METHOD M_GetAbsPos : ST_3DPoint
VAR_INPUT
	pChildPos	: POINTER TO ST_3DPoint;
	eTargetRef 	: E_TargetRef;
	nParam1		: UINT;
 	nParam2		: UINT;
	nParam3		: USINT;
	nParam4		: USINT;
	nZLevel		: USINT;
END_VAR
VAR_OUTPUT
	nErrorId 	: ERRORID;
	lrAngle		: LREAL;
END_VAR
VAR
	stLocPos : ST_3DPoint;
END_VAR
IF eTargetRef = E_TargetRef.TARGETREF_TwoDimArray THEN
	stLocPos := P_stRelPosLB;
	
	IF nParam3 = 1 THEN	//Area1
		IF nArea1CountPoints = 0 THEN
			nErrorId := E_ErrorIdObjMgmt.ERRORID_InvalidDrypadArea;  //Error
			RETURN;
		END_IF
		//X-Position berechnen
		stLocPos.X := stLocPos.X + stArea1Point1.X + (stArea1Point2.X - stArea1Point1.X) / (nArea1IntermedPointsX + 1) * (nParam1 - 1);
		//Y-Position berechnen
		stLocPos.Y := stLocPos.Y + stArea1Point1.Y + (stArea1Point2.Y - stArea1Point1.Y) / (nArea1IntermedPointsY + 1) * (nParam2 - 1);		
	ELSIF nParam3 = 2 THEN	//Area2
		IF nArea2CountPoints = 0 THEN
			nErrorId := E_ErrorIdObjMgmt.ERRORID_InvalidDrypadArea;  //Error
			RETURN;
		END_IF
		//X-Position berechnen
		stLocPos.X := stLocPos.X + stArea2Point1.X + (stArea2Point2.X - stArea2Point1.X) / (nArea2IntermedPointsX + 1) * (nParam1 - 1);
		//Y-Position berechnen
		stLocPos.Y := stLocPos.Y + stArea2Point1.Y + (stArea2Point2.Y - stArea2Point1.Y) / (nArea2IntermedPointsY + 1) * (nParam2 - 1);		
	END_IF
	
	M_GetAbsPos := pParentTarget^.M_GetAbsPos(pChildPos := ADR(stLocPos), eTargetRef:= E_TargetRef.TARGETREF_LeftBottom,
													nParam1:= 0,
													nParam2:= 0, nParam3:= 0, nParam4:= 0, nZLevel:= 0,
													lrAngle => lrAngle, nErrorId=> nErrorId);
ELSE
	M_GetAbsPos := SUPER^.M_GetAbsPos(pChildPos := pChildPos, eTargetRef:= eTargetRef,
													nParam1:= nParam1,
													nParam2:= nParam2, nParam3:= nParam3, nParam4:= 0, nZLevel:= nZLevel,
													lrAngle => lrAngle, nErrorId=> nErrorId);	
END_IF
END_METHOD

METHOD M_GetAllProps : ERRORID
VAR_INPUT
	refCmdData : REFERENCE TO  ST_CmdData;
END_VAR
SUPER^.M_GetAllProps(refCmdData);
refCmdData.aHeader[2] := nNotifyId;

nCurrentPropIndex := nCurrentPropIndex + 1;
refCmdData.n32Data[nCurrentPropIndex] := REAL_TO_DINT(rZOffset);
nCurrentPropIndex := nCurrentPropIndex + 1;
refCmdData.n32Data[nCurrentPropIndex] := REAL_TO_DINT(stArea1Point1.X);
nCurrentPropIndex := nCurrentPropIndex + 1;
refCmdData.n32Data[nCurrentPropIndex] := REAL_TO_DINT(stArea1Point1.Y);
nCurrentPropIndex := nCurrentPropIndex + 1;
refCmdData.n32Data[nCurrentPropIndex] := REAL_TO_DINT(stArea1Point2.X);
nCurrentPropIndex := nCurrentPropIndex + 1;
refCmdData.n32Data[nCurrentPropIndex] := REAL_TO_DINT(stArea1Point2.Y);
nCurrentPropIndex := nCurrentPropIndex + 1;
refCmdData.n32Data[nCurrentPropIndex] := nArea1IntermedPointsX;
nCurrentPropIndex := nCurrentPropIndex + 1;
refCmdData.n32Data[nCurrentPropIndex] := nArea1IntermedPointsY;
nCurrentPropIndex := nCurrentPropIndex + 1;
refCmdData.n32Data[nCurrentPropIndex] := REAL_TO_DINT(stArea2Point1.X);
nCurrentPropIndex := nCurrentPropIndex + 1;
refCmdData.n32Data[nCurrentPropIndex] := REAL_TO_DINT(stArea2Point1.Y);
nCurrentPropIndex := nCurrentPropIndex + 1;
refCmdData.n32Data[nCurrentPropIndex] := REAL_TO_DINT(stArea2Point2.X);
nCurrentPropIndex := nCurrentPropIndex + 1;
refCmdData.n32Data[nCurrentPropIndex] := REAL_TO_DINT(stArea2Point2.Y);
nCurrentPropIndex := nCurrentPropIndex + 1;
refCmdData.n32Data[nCurrentPropIndex] := nArea2IntermedPointsX;
nCurrentPropIndex := nCurrentPropIndex + 1;
refCmdData.n32Data[nCurrentPropIndex] := nArea2IntermedPointsY;
nCurrentPropIndex := nCurrentPropIndex + 1;
refCmdData.n32Data[nCurrentPropIndex] := nGCodeTargetNr;
END_METHOD

METHOD M_ResetPosData
VAR_INPUT
END_VAR
nCurrentColArea1 := 0;
nCurrentRowArea1 := 0;
nCurrentColArea2 := 0;
nCurrentRowArea2 := 0;
END_METHOD

METHOD M_SetAllProps : ERRORID
VAR_INPUT
	refCmdData : REFERENCE TO  ST_CmdData;
END_VAR
//Basisproperties schreiben (0 bis 7)
M_SetAllProps := SUPER^.M_SetAllProps(refCmdData);

IF M_SetAllProps > 0 THEN	//Error beim setzen der Base-Parameter
	RETURN;
END_IF

nCurrentPropIndex := nCurrentPropIndex + 1;
nSpecPropIndex := nCurrentPropIndex; 
rZOffset := DINT_TO_REAL(refCmdData.n32Data[nCurrentPropIndex]);
nCurrentPropIndex := nCurrentPropIndex + 1;
stArea1Point1.X := DINT_TO_REAL(refCmdData.n32Data[nCurrentPropIndex]);
nCurrentPropIndex := nCurrentPropIndex + 1;
stArea1Point1.Y	:= DINT_TO_REAL(refCmdData.n32Data[nCurrentPropIndex]);
nCurrentPropIndex := nCurrentPropIndex + 1;
stArea1Point2.X := DINT_TO_REAL(refCmdData.n32Data[nCurrentPropIndex]);
nCurrentPropIndex := nCurrentPropIndex + 1;
stArea1Point2.Y := DINT_TO_REAL(refCmdData.n32Data[nCurrentPropIndex]);
nCurrentPropIndex := nCurrentPropIndex + 1;
nArea1IntermedPointsX := DINT_TO_UINT(refCmdData.n32Data[nCurrentPropIndex]);
nCurrentPropIndex := nCurrentPropIndex + 1;
nArea1IntermedPointsY := DINT_TO_UINT(refCmdData.n32Data[nCurrentPropIndex]);

nArea1CountPoints := (nArea1IntermedPointsX + 2) * (nArea1IntermedPointsY + 2);

nCurrentPropIndex := nCurrentPropIndex + 1; 
stArea2Point1.X	:= DINT_TO_REAL(refCmdData.n32Data[nCurrentPropIndex]);
nCurrentPropIndex := nCurrentPropIndex + 1;
stArea2Point1.Y	:= DINT_TO_REAL(refCmdData.n32Data[nCurrentPropIndex]);
nCurrentPropIndex := nCurrentPropIndex + 1;
stArea2Point2.X	:= DINT_TO_REAL(refCmdData.n32Data[nCurrentPropIndex]);
nCurrentPropIndex := nCurrentPropIndex + 1;
stArea2Point2.Y	:= DINT_TO_REAL(refCmdData.n32Data[nCurrentPropIndex]);
nCurrentPropIndex := nCurrentPropIndex + 1;
nArea2IntermedPointsX := DINT_TO_UINT(refCmdData.n32Data[nCurrentPropIndex]);
nCurrentPropIndex := nCurrentPropIndex + 1;
nArea2IntermedPointsY := DINT_TO_UINT(refCmdData.n32Data[nCurrentPropIndex]);

IF stArea2Point1.X <  stArea2Point2.X AND stArea2Point1.Y <  stArea2Point2.Y THEN
	nArea2CountPoints := (nArea2IntermedPointsX + 2) * (nArea2IntermedPointsY + 2);
ELSE
 	nArea2CountPoints := 0;
END_IF

nCurrentPropIndex := nCurrentPropIndex + 1;
nGCodeTargetNr := DINT_TO_UINT(refCmdData.n32Data[nCurrentPropIndex]);
nNoOfProps := nCurrentPropIndex + 1;
END_METHOD

METHOD M_SetSingleProp : ERRORID
VAR_INPUT
	refCmdData : REFERENCE TO  ST_CmdData;
END_VAR
IF nSpecPropIndex = refCmdData.aHeader[1] THEN
	rZOffset := DINT_TO_REAL(refCmdData.n32Data[0]);
ELSIF (nSpecPropIndex + 1) = refCmdData.aHeader[1] THEN
	stArea1Point1.X := DINT_TO_REAL(refCmdData.n32Data[0]);
ELSIF (nSpecPropIndex + 2) = refCmdData.aHeader[1] THEN
	stArea1Point1.Y := DINT_TO_REAL(refCmdData.n32Data[0]);
ELSIF (nSpecPropIndex + 3) = refCmdData.aHeader[1] THEN
	stArea1Point2.X := DINT_TO_REAL(refCmdData.n32Data[0]);
ELSIF (nSpecPropIndex + 4) = refCmdData.aHeader[1] THEN
	stArea1Point2.Y := DINT_TO_REAL(refCmdData.n32Data[0]);
ELSIF (nSpecPropIndex + 5) = refCmdData.aHeader[1] THEN
	nArea1IntermedPointsX := DINT_TO_UINT(refCmdData.n32Data[0]);
ELSIF (nSpecPropIndex + 6) = refCmdData.aHeader[1] THEN
	nArea1IntermedPointsY := DINT_TO_UINT(refCmdData.n32Data[0]);
ELSIF (nSpecPropIndex + 7) = refCmdData.aHeader[1] THEN
	stArea2Point1.X := DINT_TO_REAL(refCmdData.n32Data[0]);
ELSIF (nSpecPropIndex + 8) = refCmdData.aHeader[1] THEN
	stArea2Point1.Y := DINT_TO_REAL(refCmdData.n32Data[0]);
ELSIF (nSpecPropIndex + 9) = refCmdData.aHeader[1] THEN
	stArea2Point2.X := DINT_TO_REAL(refCmdData.n32Data[0]);
ELSIF (nSpecPropIndex + 10) = refCmdData.aHeader[1] THEN
	stArea2Point2.Y := DINT_TO_REAL(refCmdData.n32Data[0]);
ELSIF (nSpecPropIndex + 11) = refCmdData.aHeader[1] THEN
	nArea2IntermedPointsX := DINT_TO_UINT(refCmdData.n32Data[0]);
ELSIF (nSpecPropIndex + 12) = refCmdData.aHeader[1] THEN
	nArea2IntermedPointsY := DINT_TO_UINT(refCmdData.n32Data[0]);
ELSE
	M_SetSingleProp := SUPER^.M_SetSingleProp(refCmdData);
END_IF
END_METHOD

METHOD M_UpdateProcessData
VAR_INPUT
END_VAR
//Processdaten übetragen
aObjProcData[nNotifyId].nObjId := nObjectID;
aObjProcData[nNotifyId].n32Data[0] := nArea1CountPoints;
IF nCurrentColArea1 = 0 THEN
	aObjProcData[nNotifyId].n32Data[1] := 0;
ELSE
	aObjProcData[nNotifyId].n32Data[1] := (nArea1IntermedPointsX + 2) * (nCurrentRowArea1 - 1) + nCurrentColArea1;
END_IF

aObjProcData[nNotifyId].n32Data[2] := nArea2CountPoints;

IF nCurrentColArea2 = 0 THEN
	aObjProcData[nNotifyId].n32Data[3] := 0;
ELSE
	aObjProcData[nNotifyId].n32Data[3] := (nArea2IntermedPointsX + 2) * (nCurrentRowArea2 - 1) + nCurrentColArea2;
END_IF
END_METHOD

PROPERTY P_nGCodeTargetNr : UINT
GET
P_nGCodeTargetNr := nGCodeTargetNr;
END_GET
END_PROPERTY

PROPERTY P_nNotifyId : UINT
GET
P_nNotifyId := nNotifyId;
END_GET
SET
nNotifyId := P_nNotifyId;
END_SET
END_PROPERTY

END_FUNCTION_BLOCK

// ---- Objects/Targets/Active/FB_TipCleaner.TcPOU
FUNCTION_BLOCK FB_TipCleaner EXTENDS FB_ActiveTarget
VAR
	eBasicAction		: E_Action;
	eStripState			: E_OpClState;
	
	//Spec-Properties
	stFirstPoint		: ST_3DPoint;	//FirstPoint und LastPoint ergeben eine Linie
	stLastPoint			: ST_3DPoint;	//FirstPoint und LastPoint ergeben eine Linie
	nIntermedPoints		: USINT;		//Anzahl der Punkte auf der von FirstPoint und LastPoint gebildeten Linie
	
	nClosedPos			: UINT;			//Verschlussposition
	
	//****************************************Aktionvariablen****************************************************
	bActionLock			: ARRAY[50..150] OF BOOL;
	
	fbTipCleanerInit	: FB_TipCleanerInit;
	
	//Action: "OpenClose"
	bOpenClose			: BOOL;
	nStateA_OpenClose	: USINT;	//Statemachine von A_OpenClose();
	nOpenCloseMode		: USINT;	//0=Open, 1=Close

END_VAR

VAR PERSISTENT
	nCurrentPoint		: USINT;
END_VAR

IF bInitFB THEN
	bInitFB := FALSE;
	F_CreateLinkedListHnd( ADR( aNodes ), SIZEOF( aNodes ), hList );
	//Fehlerstruktur vorausfüllen
	stError.ObjectId := nObjectID;
	stError.HardwareGrp := E_HardwareGrp.Nothing;
	stError.POU := E_POU.POU_FB_TipCleaner;
END_IF

CASE eCurrentState OF
	E_MachineState.MACHINESTATE_Active:
		//BasicActions ausführen
		IF bInit THEN	//Initialisieren
			A_Init();
			IF nStateA_Init >= 80 THEN
				bIsInit := TRUE;
				IF nStateA_Init >= 99 THEN
					bError := TRUE;
					bIsInit := FALSE;	
				END_IF
				bInit := FALSE;
				nStateA_Init := 0;
				M_RemoveListEntry(nSearchValue:= E_Action.ACTION_Init);
			END_IF
		END_IF
		
		IF bOpenClose THEN	//Backen auf/zu
			A_OpenClose();
			IF nStateA_OpenClose >= 80 THEN
				IF nStateA_OpenClose >= 99 THEN
					bError := TRUE;	
				END_IF
				bOpenClose := FALSE;
				nStateA_OpenClose := 0;
				M_RemoveListEntry(nSearchValue:= E_Action.ACTION_OpenClose);
			END_IF
		END_IF		

		IF hList.nCount = 0 THEN
			eCurrentState := E_MachineState.MACHINESTATE_Ready;
		END_IF

		IF bError  THEN
			eCurrentState := E_MachineState.MACHINESTATE_Error;
		END_IF		
	
	E_MachineState.MACHINESTATE_Reset:
		A_Reset();
		IF nStateA_Reset = 80 THEN
			nStateA_Init := 0;
			nStateA_OpenClose := 0;
			nStateA_Stop := 0;
			nStateA_Reset := 0;
			bBusy := FALSE;
			bError := FALSE;
			bStopAllOnError := FALSE;
			fbList.A_Reset(hList := hList);
			MEMSET(ADR(bActionLock),0,SIZEOF(bActionLock));
			nErrorId := 0;
			stError.Cmd := 0;
			stError.ErrorId := 0;
			eCurrentState := E_MachineState.MACHINESTATE_Idle;
		ELSIF
			nStateA_Reset = 99 THEN
			fbErrorList.M_Add(stError);
			nStateA_Reset := 0;
			bBusy := FALSE;
			bError := TRUE;
			eCurrentState := E_MachineState.MACHINESTATE_Error;			
		END_IF
	
	E_MachineState.MACHINESTATE_Ready:
		bBusy := FALSE;
		eCurrentState := E_MachineState.MACHINESTATE_Idle;
		
	E_MachineState.MACHINESTATE_Error:
		bBusy := FALSE;	
	
END_CASE

//Prozessdaten aktualisieren
stProcessData.nObjId := nObjectID;
stProcessData.n32Data[0] := BOOL_TO_DINT(bIsInit);
stProcessData.n32Data[1] := eCurrentState;
stProcessData.n32Data[2] := stError.ErrorId;
IF stTipCleanerRef.nCurrentPos = 0 THEN
	eStripState := E_OpClState.Open;
	stProcessData.n32Data[3] := E_OpClState.Open;
ELSIF stTipCleanerRef.nCurrentPos = nClosedPos THEN
		eStripState := E_OpClState.Closed;
	stProcessData.n32Data[3] := E_OpClState.Closed;
ELSE
	eStripState := E_OpClState.UNDEFINED;
	stProcessData.n32Data[3] := E_OpClState.UNDEFINED;
END_IF

stProcessData.n32Data[4] := nIntermedPoints + 2; //Konfigurierte Reinigungspositionen
stProcessData.n32Data[5] := nCurrentPoint;	//verbrauchte Reinigungspositionen

aObjProcData[nNotifyId] := stProcessData;

ACTION A_Init:
IF nStateA_Init = 0 THEN
	bIsInit := FALSE;

	IF bFlagA_Init XOR fbTipCleanerInit.bBusy  THEN
		bFlagA_Init := FALSE;
		fbTipCleanerInit(pstTipCleanerRef:= ADR(stTipCleanerRef), bExecute:= TRUE);
	ELSE
		RETURN;	//damit nachfolgende Zeilen nicht bearbeitet werden
	END_IF		

	IF NOT fbTipCleanerInit.bBusy THEN
		IF fbTipCleanerInit.bError THEN
			stError.ErrorId := fbTipCleanerInit.nErrorId;
			stError.POUState := nStateA_Init;
			nStateA_Init := 99;
		ELSE
			bFlagA_Init := TRUE;
			nStateA_Init := 80;
		END_IF
		fbTipCleanerInit(pstTipCleanerRef:= ADR(stTipCleanerRef), bExecute:= FALSE);
	END_IF
END_IF

//Errorhandling
IF nStateA_Init = 99 THEN
	stError.Cmd := E_Action.ACTION_Init;
	stError.POUAction := E_POUACT.POUACT_A_Init;
	fbErrorList.M_Add(stError);
END_IF
END_ACTION

ACTION A_OpenClose:
stError.POUState := nStateA_OpenClose;

IF stTipCleanerRef.nStatus.3 THEN	//Error
	stError.ErrorId := E_ErrorIdCmd.ERRORID_DeviceInErrorState;
	nStateA_OpenClose := 99;
END_IF

CASE nStateA_OpenClose OF
	0:
		IF nOpenCloseMode = 0 THEN	//Öffnen
			stTipCleanerRef.nTargetPos := 0;
		ELSE	//Schließen
			stTipCleanerRef.nTargetPos := nClosedPos;
		END_IF
		
		stTipCleanerRef.nControl := 31;
		
		IF stTipCleanerRef.nStatus.12 THEN	//Setpoint acknowledge
			stTipCleanerRef.nControl := 15;
			nStateA_OpenClose := 1;
		END_IF
		
	1:	//Warten auf Target reached
		IF stTipCleanerRef.nStatus.10 THEN	//Target reached
			nStateA_OpenClose := 80;
		END_IF
		
	70:	//Cancel
		nStateA_OpenClose := 80;
END_CASE

//Errorhandling
IF nStateA_OpenClose = 99 THEN
	stError.Cmd := E_Action.ACTION_OpenClose;
	stError.POUAction := E_POUACT.POUACT_A_OpenClose;
	fbErrorList.M_Add(stError);
END_IF
END_ACTION

ACTION A_Reset:
CASE nStateA_Reset OF
	0:
		nStateA_Reset := 80;
END_CASE
END_ACTION

METHOD FB_init : BOOL
VAR_INPUT
	bInitRetains : BOOL; // if TRUE, the retain variables are initialized (warm start / cold start)
	bInCopyCode : BOOL;  // if TRUE, the instance afterwards gets moved into the copy code (online change)
END_VAR
eObjectType := E_ObjectType.OBJECTTYPE_TipCleaner;
eObjectGroup := E_ObjectGroup.OBJECTGROUP_Target OR E_ObjectGroup.OBJECTGROUP_Device;
END_METHOD

METHOD M_ChangeCleanMat
VAR_INPUT
END_VAR
nCurrentPoint := 0;
END_METHOD

METHOD M_CheckAction : ERRORID
VAR_INPUT
	refActionData 	: REFERENCE TO ST_ActionData;
	pCorrelObject	: POINTER TO FB_Object;
END_VAR
IF NOT refActionData.eAction = E_Action.ACTION_MoveToTarget THEN
	M_CheckAction := 8989;	
END_IF
END_METHOD

METHOD M_CheckProcDataType : BOOL
VAR_INPUT
	eProcDataType : E_ProcDataType;
END_VAR
END_METHOD

METHOD M_ExeAction : ERRORID
VAR_INPUT
	refActionData : REFERENCE TO ST_ActionData;	
END_VAR
IF NOT (eCurrentState = E_MachineState.MACHINESTATE_Idle OR
	eCurrentState = E_MachineState.MACHINESTATE_Active OR
	eCurrentState = E_MachineState.MACHINESTATE_Ready) THEN
	M_ExeAction := E_ErrorIdCmd.ERRORID_InvalidState;
	RETURN;
END_IF

CASE refActionData.eAction OF
	E_Action.ACTION_Init:
		IF NOT bInit THEN
			bInit := TRUE;
			fbList.A_AddHeadValue(hList := hList, putValue:= E_Action.ACTION_Init);
		ELSE
			RETURN;
		END_IF
		
	E_Action.ACTION_OpenClose:
		IF NOT bOpenClose THEN
			IF NOT bIsInit THEN
				M_ExeAction := E_ErrorIdCmd.ERRORID_DeviceNotInitialized;  //Error
				RETURN;
			END_IF
			nOpenCloseMode := DINT_TO_USINT(refActionData.aParams[1]);
			fbList.A_AddHeadValue(hList := hList, putValue:= E_Action.ACTION_OpenClose);
			bOpenClose := TRUE;
		ELSE
			RETURN;
		END_IF
		
	E_Action.ACTION_Stop:
		//Stop braucht nur ausgeführt werden, wenn irgendwas aktiv ist
		fbList.A_AddHeadValue(hList := hList, putValue:= E_Action.ACTION_Stop);		
	ELSE
		M_ExeAction := E_ErrorIdCmd.ERRORID_InvalidAction;
END_CASE
bBusy := TRUE;
eCurrentState := E_MachineState.MACHINESTATE_Active;
END_METHOD

METHOD M_GetAbsPos : ST_3DPoint
VAR_INPUT
	pChildPos	: POINTER TO ST_3DPoint;
	eTargetRef 	: E_TargetRef;
	nParam1		: UINT;
 	nParam2		: UINT;
	nParam3		: USINT;
	nParam4		: USINT;
	nZLevel		: USINT;
END_VAR
VAR_OUTPUT
	nErrorId 	: ERRORID;
	lrAngle		: LREAL;
END_VAR
VAR
	stLocPosLB : ST_3DPoint;
	rSpace	: REAL;
END_VAR
IF eTargetRef = E_TargetRef.TARGETREF_SpecPoint THEN
	stLocPosLB := P_stRelPosLB;
	IF nParam1 = 1 THEN
		stLocPosLB := F_Add3DPoints(stLocPosLB,stFirstPoint);
	ELSIF nParam1 = 2 THEN
		stLocPosLB := F_Add3DPoints(stLocPosLB,stLastPoint);
	ELSE
		nErrorId := E_ErrorIdCmd.ERRORID_InvalidTargetPointNr;
		RETURN;
	END_IF
	M_GetAbsPos := pParentTarget^.M_GetAbsPos(pChildPos := ADR(stLocPosLB), eTargetRef:= E_TargetRef.TARGETREF_LeftBottom,
												nParam1:= 0,
												nParam2:= 0, nParam3:= 0, nParam4:= 0, nZLevel:= 0,
												lrAngle => lrAngle, nErrorId=> nErrorId);	
ELSIF eTargetRef = E_TargetRef.TARGETREF_TwoDimArray THEN
	//Checken ob gültiger Punkt
	IF nParam1 = 0 OR nParam1 > (nIntermedPoints + 2) THEN
		nErrorId := E_ErrorIdCmd.ERRORID_InvalidTargetPointCol;
		RETURN;
	END_IF
	stLocPosLB := P_stRelPosLB;
	//Ausrichtung in X oder Y?
	IF stFirstPoint.Y = stLastPoint.Y THEN	//Ausrichtung in X
		//X-Position berechnen
		//Space(Zwischenräume zwischen den Punkten berechnen
		rSpace := (stLastPoint.X - stFirstPoint.X) / (nIntermedPoints + 1); 
		stLocPosLB.X := stLocPosLB.X + stFirstPoint.X + (nParam1 - 1) * rSpace;
		//Y-Position berechenen
		stLocPosLB.Y := stLocPosLB.Y + stFirstPoint.Y;
	ELSIF stFirstPoint.X = stLastPoint.X THEN //Ausrichtung in Y
		//X-Position berechnen
		stLocPosLB.X := stLocPosLB.X + stFirstPoint.X;
		//Y-Position berechenen
		//Space(Zwischenräume zwischen den Punkten berechnen
		rSpace := (stLastPoint.Y - stFirstPoint.Y) / (nIntermedPoints + 1);
		stLocPosLB.Y := stLocPosLB.Y + stFirstPoint.Y + (nParam1 - 1) * rSpace;
	ELSE
		nErrorId := E_ErrorIdCmd.ERRORID_InvalidTargetPointCol;
		RETURN;
	END_IF
	stLocPosLB.Z := stLocPosLB.Z + stFirstPoint.Z;
	M_GetAbsPos := pParentTarget^.M_GetAbsPos(pChildPos := ADR(stLocPosLB), eTargetRef:= E_TargetRef.TARGETREF_LeftBottom,
												nParam1:= 0,
												nParam2:= 0, nParam3:= 0,nParam4:= 0, nZLevel:= 0,
												lrAngle => lrAngle, nErrorId=> nErrorId);	

ELSE
	M_GetAbsPos := SUPER^.M_GetAbsPos(pChildPos := pChildPos, eTargetRef:= eTargetRef,
													nParam1:= nParam1,
													nParam2:= nParam2, nParam3:= nParam3, nParam4:= 0, nZLevel:= nZLevel,
													lrAngle => lrAngle, nErrorId=> nErrorId);	
END_IF
END_METHOD

METHOD M_GetActionBusy : BOOL
VAR_INPUT
	eAction : E_Action;
END_VAR
getPosPtr := 0;(* start from first node element *)
fbList.A_FindNext( hList := hList, putPosPtr := getPosPtr, putValue := eAction, getValue=>getValue, getPosPtr=>getPosPtr );
IF fbList.bOk THEN	//Eintrag wurde gefunden, d.h. Action ist noch busy
	M_GetActionBusy := TRUE;
END_IF
END_METHOD

METHOD M_GetAllProps : ERRORID
VAR_INPUT
	refCmdData : REFERENCE TO  ST_CmdData;
END_VAR
SUPER^.M_GetAllProps(refCmdData);
nCurrentPropIndex := nCurrentPropIndex + 1;
refCmdData.n32Data[nCurrentPropIndex] := REAL_TO_DINT(stFirstPoint.X);
nCurrentPropIndex := nCurrentPropIndex + 1;
refCmdData.n32Data[nCurrentPropIndex] := REAL_TO_DINT(stFirstPoint.Y);
nCurrentPropIndex := nCurrentPropIndex + 1;
refCmdData.n32Data[nCurrentPropIndex] := REAL_TO_DINT(stFirstPoint.Z);
nCurrentPropIndex := nCurrentPropIndex + 1;
refCmdData.n32Data[nCurrentPropIndex] := REAL_TO_DINT(stLastPoint.X);
nCurrentPropIndex := nCurrentPropIndex + 1;
refCmdData.n32Data[nCurrentPropIndex] := REAL_TO_DINT(stLastPoint.Y);
nCurrentPropIndex := nCurrentPropIndex + 1;
refCmdData.n32Data[nCurrentPropIndex] := nIntermedPoints;
nCurrentPropIndex := nCurrentPropIndex + 1;
refCmdData.n32Data[nCurrentPropIndex] := nClosedPos;
END_METHOD

METHOD M_GetNextPointNr : USINT
VAR_INPUT
END_VAR
IF (nCurrentPoint = (nIntermedPoints + 2)) OR (nCurrentPoint = 0) THEN
	nCurrentPoint := 1;
ELSE
	nCurrentPoint := nCurrentPoint + 1;
END_IF
M_GetNextPointNr := nCurrentPoint;
END_METHOD

METHOD M_GetProcData : DINT
VAR_INPUT
	eProcDataType : E_ProcDataType;
END_VAR
END_METHOD

METHOD M_RemoveListEntry : BOOL
VAR_INPUT
	nSearchValue	: E_Action;
END_VAR
getPosPtr := 0;(* start from first node element *)
fbList.A_FindNext( hList := hList, putPosPtr := getPosPtr, putValue := nSearchValue, getValue=>getValue, getPosPtr=>getPosPtr );
IF fbList.bOk THEN	//Eintrag wurde gefunden
	fbList.A_RemoveValueAtPosPtr(hList:= hList,	putPosPtr:= getPosPtr);
	IF fbList.bOk THEN
		M_RemoveListEntry := TRUE;
	END_IF
END_IF
END_METHOD

METHOD M_SetAllProps : ERRORID
VAR_INPUT
	refCmdData : REFERENCE TO  ST_CmdData;
END_VAR
M_SetAllProps := SUPER^.M_SetAllProps(refCmdData);

IF M_SetAllProps > 0 THEN
	RETURN;
END_IF

nCurrentPropIndex := nCurrentPropIndex + 1;
nSpecPropIndex := nCurrentPropIndex;
stFirstPoint.X := DINT_TO_REAL(refCmdData.n32Data[nCurrentPropIndex]);
nCurrentPropIndex := nCurrentPropIndex + 1;
stFirstPoint.Y := DINT_TO_REAL(refCmdData.n32Data[nCurrentPropIndex]);
nCurrentPropIndex := nCurrentPropIndex + 1;
stFirstPoint.Z := DINT_TO_REAL(refCmdData.n32Data[nCurrentPropIndex]);
nCurrentPropIndex := nCurrentPropIndex + 1; 
stLastPoint.X := DINT_TO_REAL(refCmdData.n32Data[nCurrentPropIndex]);
nCurrentPropIndex := nCurrentPropIndex + 1;
stLastPoint.Y := DINT_TO_REAL(refCmdData.n32Data[nCurrentPropIndex]);
stLastPoint.Z := stFirstPoint.Z;
nCurrentPropIndex := nCurrentPropIndex + 1;
nIntermedPoints := DINT_TO_USINT(refCmdData.n32Data[nCurrentPropIndex]);
nCurrentPropIndex := nCurrentPropIndex + 1;
nClosedPos := DINT_TO_UINT(refCmdData.n32Data[nCurrentPropIndex]);

nNoOfProps := nCurrentPropIndex + 1;
END_METHOD

METHOD M_SetSingleProp : ERRORID
VAR_INPUT
	refCmdData : REFERENCE TO  ST_CmdData;
END_VAR
IF nSpecPropIndex = refCmdData.aHeader[1] THEN
	stFirstPoint.X := DINT_TO_REAL(refCmdData.n32Data[0]);
ELSIF (nSpecPropIndex + 1) = refCmdData.aHeader[1] THEN
	stFirstPoint.Y := DINT_TO_REAL(refCmdData.n32Data[0]);
ELSIF (nSpecPropIndex + 2) = refCmdData.aHeader[1] THEN
	stFirstPoint.Z := DINT_TO_REAL(refCmdData.n32Data[0]);
ELSIF (nSpecPropIndex + 3) = refCmdData.aHeader[1] THEN
	stLastPoint.X := DINT_TO_REAL(refCmdData.n32Data[0]);
ELSIF (nSpecPropIndex + 4) = refCmdData.aHeader[1] THEN
	stLastPoint.Y := DINT_TO_REAL(refCmdData.n32Data[0]);
ELSIF (nSpecPropIndex + 5) = refCmdData.aHeader[1] THEN
	nIntermedPoints := DINT_TO_USINT(refCmdData.n32Data[0]);
ELSIF (nSpecPropIndex + 6) = refCmdData.aHeader[1] THEN
	nClosedPos := DINT_TO_UINT(refCmdData.n32Data[0]);	
ELSE
	M_SetSingleProp := SUPER^.M_SetSingleProp(refCmdData);
END_IF
END_METHOD

METHOD M_Stop : ERRORID
VAR_INPUT
END_VAR
IF bOpenClose THEN
	nStateA_OpenClose := 70;
END_IF
END_METHOD

PROPERTY P_eStripState : E_OpClState
GET
P_eStripState := eStripState;
END_GET
END_PROPERTY

END_FUNCTION_BLOCK

// ---- Hardware/TipCleaner/FB_TipCleanerInit.TcPOU
FUNCTION_BLOCK FB_TipCleanerInit
VAR_INPUT
	pstTipCleanerRef	: POINTER TO ST_TipCleanerRef;
	bExecute			: BOOL;
END_VAR
VAR_OUTPUT
	bBusy		: BOOL;
	bError		: BOOL;
	nErrorId	: ERRORID;
END_VAR
VAR
	fbSdoWrite	: FB_SDO_WRITE;
	nIndex		: DWORD;
	nSubIndex	: DWORD;
	nDataLength	: DWORD;
	nData		: DINT;
	nState		: USINT;
	timer		: TON;
END_VAR

IF bExecute THEN
	bBusy := TRUE;
	CASE nState OF
		0:	//*************ANFANG INITIALISIERUNG ************************************
			IF pstTipCleanerRef^.nStatus.3 THEN	//Error?
				pstTipCleanerRef^.nControl := 153;	//Error zurücksetzen
			ELSE
				pstTipCleanerRef^.nControl := 0;
				nState := nState + 1;
			END_IF
			
		1:	//max Strom auf 0,8A begrenzen (TMCM1140 max 2A entspricht "255" in Object 0x2003)
			fbSdoWrite(sADSNetID:= pstTipCleanerRef^.stAdsAdress.sNetId,nPortNr:= pstTipCleanerRef^.stAdsAdress.nPort, 
						nIndex:= 16#2003, nSubIndex:= 0, nDataLength:= 1, nData:= 128, bExecute:= TRUE);
			 	
			IF NOT fbSdoWrite.bBusy THEN
				IF fbSdoWrite.bError THEN
					nErrorId := fbSdoWrite.nAdsErrorId;
					nState := 99;
				ELSE
					nState := nState + 1;
				END_IF
				fbSdoWrite(bExecute:= FALSE);
			END_IF

		2:	//Standby Strom auf 0,2A begrenzen (TMCM1140 max 2A entspricht "255" in Object 0x2004)
			(*fbSdoWrite(sADSNetID:= pstTipCleanerRef^.stAdsAdress.sNetId,nPortNr:= pstTipCleanerRef^.stAdsAdress.nPort, 
						nIndex:= 16#2004, nSubIndex:= 0, nDataLength:= 1, nData:= 35, bExecute:= TRUE);*)
			 	
			fbSdoWrite(sADSNetID:= pstTipCleanerRef^.stAdsAdress.sNetId,nPortNr:= pstTipCleanerRef^.stAdsAdress.nPort, 
						nIndex:= 16#2004, nSubIndex:= 0, nDataLength:= 1, nData:= 0, bExecute:= TRUE);

			IF NOT fbSdoWrite.bBusy THEN
				IF fbSdoWrite.bError THEN
					nErrorId := fbSdoWrite.nAdsErrorId;
					nState := 99;
				ELSE
					nState := nState + 1;
				END_IF
				fbSdoWrite(bExecute:= FALSE);
			END_IF
			
		3:	//SwitchParameters setzen (keine Endlagen verwenden)
			fbSdoWrite(sADSNetID:= pstTipCleanerRef^.stAdsAdress.sNetId,nPortNr:= pstTipCleanerRef^.stAdsAdress.nPort, 
						nIndex:= 16#2005, nSubIndex:= 0, nDataLength:= 4, nData:= 3, bExecute:= TRUE);
			 	
			IF NOT fbSdoWrite.bBusy THEN
				IF fbSdoWrite.bError THEN
					nErrorId := fbSdoWrite.nAdsErrorId;
					nState := 99;
				ELSE
					nState := nState + 1;
				END_IF
				fbSdoWrite(bExecute:= FALSE);
			END_IF

		4:	//Brake deaktivieren
			fbSdoWrite(sADSNetID:= pstTipCleanerRef^.stAdsAdress.sNetId,nPortNr:= pstTipCleanerRef^.stAdsAdress.nPort, 
						nIndex:= 16#200C, nSubIndex:= 2, nDataLength:= 1, nData:= 0, bExecute:= TRUE);

			IF NOT fbSdoWrite.bBusy THEN
				IF fbSdoWrite.bError THEN
					nErrorId := fbSdoWrite.nAdsErrorId;
					nState := 99;
				ELSE
					nState := nState + 1;
				END_IF
				fbSdoWrite(bExecute:= FALSE);
			END_IF
			
		5:	//Digital Outputmask setzen
			fbSdoWrite(sADSNetID:= pstTipCleanerRef^.stAdsAdress.sNetId,nPortNr:= pstTipCleanerRef^.stAdsAdress.nPort, 
						nIndex:= 16#2703, nSubIndex:= 2, nDataLength:= 4, nData:= 16#30000, bExecute:= TRUE);

			IF NOT fbSdoWrite.bBusy THEN
				IF fbSdoWrite.bError THEN
					nErrorId := fbSdoWrite.nAdsErrorId;
					nState := 99;
				ELSE
					nState := nState + 1;
				END_IF
				fbSdoWrite(bExecute:= FALSE);
			END_IF

		6:	//Fast Homing Speed setzen
			fbSdoWrite(sADSNetID:= pstTipCleanerRef^.stAdsAdress.sNetId,nPortNr:= pstTipCleanerRef^.stAdsAdress.nPort, 
						nIndex:= 16#6099, nSubIndex:= 1, nDataLength:= 4, nData:= 200, bExecute:= TRUE);

			IF NOT fbSdoWrite.bBusy THEN
				IF fbSdoWrite.bError THEN
					nErrorId := fbSdoWrite.nAdsErrorId;
					nState := 99;
				ELSE
					nState := nState + 1;
				END_IF
				fbSdoWrite(bExecute:= FALSE);
			END_IF

		7:	//Slow Homing Speed setzen
			fbSdoWrite(sADSNetID:= pstTipCleanerRef^.stAdsAdress.sNetId,nPortNr:= pstTipCleanerRef^.stAdsAdress.nPort, 
						nIndex:= 16#6099, nSubIndex:= 2, nDataLength:= 4, nData:= 100, bExecute:= TRUE);

			IF NOT fbSdoWrite.bBusy THEN
				IF fbSdoWrite.bError THEN
					nErrorId := fbSdoWrite.nAdsErrorId;
					nState := 99;
				ELSE
					nState := nState + 1;
				END_IF
				fbSdoWrite(bExecute:= FALSE);
			END_IF
			
		8:	//Profile Velo setzen
			fbSdoWrite(sADSNetID:= pstTipCleanerRef^.stAdsAdress.sNetId,nPortNr:= pstTipCleanerRef^.stAdsAdress.nPort, 
						nIndex:= 16#6081, nSubIndex:= 0, nDataLength:= 4, nData:= 800, bExecute:= TRUE);

			IF NOT fbSdoWrite.bBusy THEN
				IF fbSdoWrite.bError THEN
					nErrorId := fbSdoWrite.nAdsErrorId;
					nState := 99;
				ELSE
					nState := nState + 1;
				END_IF
				fbSdoWrite(bExecute:= FALSE);
			END_IF

		9:	//Homing Method setzen
			fbSdoWrite(sADSNetID:= pstTipCleanerRef^.stAdsAdress.sNetId,nPortNr:= pstTipCleanerRef^.stAdsAdress.nPort, 
						nIndex:= 16#6098, nSubIndex:= 0, nDataLength:= 1, nData:= 19, bExecute:= TRUE);

			IF NOT fbSdoWrite.bBusy THEN
				IF fbSdoWrite.bError THEN
					nErrorId := fbSdoWrite.nAdsErrorId;
					nState := 99;
				ELSE
					nState := nState + 1;
				END_IF
				fbSdoWrite(bExecute:= FALSE);
			END_IF
			
		10:	//Position Window setzen
			fbSdoWrite(sADSNetID:= pstTipCleanerRef^.stAdsAdress.sNetId,nPortNr:= pstTipCleanerRef^.stAdsAdress.nPort, 
						nIndex:= 16#6067, nSubIndex:= 0, nDataLength:= 4, nData:= 100, bExecute:= TRUE);

			IF NOT fbSdoWrite.bBusy THEN
				IF fbSdoWrite.bError THEN
					nErrorId := fbSdoWrite.nAdsErrorId;
					nState := 99;
				ELSE
					nState := nState + 1;
				END_IF
				fbSdoWrite(bExecute:= FALSE);
			END_IF
			
		11:	//Leistungsteil einschalten - "Ready to switch on"
			pstTipCleanerRef^.nControl := 6;
			pstTipCleanerRef^.bVDD5V := TRUE;	//Versorgung für Digitale IOs (5V) einschalten
			nState := nState + 1;

		12:	//Abfrage auf Status "Ready to switch on"
			IF F_GetCoDS402State(pstTipCleanerRef^.nStatus) = E_CoDS402States.DS402STATE_Fault THEN  //Error
				nState := 99;
			ELSIF F_GetCoDS402State(pstTipCleanerRef^.nStatus) = E_CoDS402States.DS402STATE_ReadyToSwitchOn  THEN//"Ready to switch on"
				nState := nState + 1;
			END_IF

		13:	//Leistungsteil einschalten - "Switch on" und "Voltage Enabled"
			pstTipCleanerRef^.nControl := 7;
			nState := nState + 1;
			
		14:	//Abfrage auf Status "Switch on" und "Voltage Enabled"
			IF F_GetCoDS402State(pstTipCleanerRef^.nStatus) = E_CoDS402States.DS402STATE_Fault THEN  //Error
				nState := 99;
			ELSIF F_GetCoDS402State(pstTipCleanerRef^.nStatus) = E_CoDS402States.DS402STATE_SwitchedOn THEN //"Switch on" und "Voltage Enabled"
				nState := nState + 1;
			END_IF

		15:	//Leistungsteil einschalten - "Operation Enabled"
			pstTipCleanerRef^.nControl := 15;
			nState := nState + 1;

		16:	//Abfrage auf Status "Operation Enabled"
			IF F_GetCoDS402State(pstTipCleanerRef^.nStatus) = E_CoDS402States.DS402STATE_Fault THEN  //Error
				nState := 99;
			ELSIF F_GetCoDS402State(pstTipCleanerRef^.nStatus) = E_CoDS402States.DS402STATE_OperationEnabled THEN //"Operation Enabled"
				nState := nState + 1;
			END_IF
			
		17:	//Mode of Operation auf "Homing" setzen
			pstTipCleanerRef^.nMode := 6;
			IF pstTipCleanerRef^.nModeDisp = 6 THEN
				nState := nState + 1;
			END_IF
			
		18:	//Homing Starten
			pstTipCleanerRef^.nControl := 31;
			IF pstTipCleanerRef^.nStatus.3 OR pstTipCleanerRef^.nStatus.13 THEN //Error
				nState := 99;
			ELSIF NOT pstTipCleanerRef^.nStatus.10 AND NOT pstTipCleanerRef^.nStatus.12 AND NOT pstTipCleanerRef^.nStatus.13 THEN	//Homig in process
				nState := nState + 1;
				timer(IN:= FALSE);
			END_IF
			
		19:	//Homing ready?
			timer(IN:= TRUE, PT:=T#6S);
			IF timer.Q THEN	//Error
				timer(IN:= FALSE);
				pstTipCleanerRef^.nControl := 0;
				nState := 99;
				RETURN;
			END_IF
			
			IF pstTipCleanerRef^.nStatus.3 OR pstTipCleanerRef^.nStatus.13 THEN //Error
				nState := 99;
			ELSIF pstTipCleanerRef^.nStatus.10 AND pstTipCleanerRef^.nStatus.12 AND NOT pstTipCleanerRef^.nStatus.13 THEN
				pstTipCleanerRef^.nControl := 15;
				nState := nState + 1;
			END_IF

		20:	//Mode of Operation auf "PP" setzen
			pstTipCleanerRef^.nMode := 1;
			IF pstTipCleanerRef^.nModeDisp = 1 THEN
				nState := nState + 1;
				bBusy := FALSE;
			END_IF

		99:	//Error
			bBusy := FALSE;
			bError := TRUE;
	END_CASE
 ELSE
	bError := FALSE;
	nErrorId := 0;
	nState := 0;
END_IF

END_FUNCTION_BLOCK

// ---- Hardware/F_GetCoDS402State.TcPOU
FUNCTION F_GetCoDS402State : E_CoDS402States
VAR_INPUT
	nStatus	: UINT;
END_VAR
VAR
	nStatusTemp	: UINT;
END_VAR

IF (nStatus AND 16#4F) = 0 THEN
	F_GetCoDS402State := E_CoDS402States.DS402STATE_NotReadyToSwitchOn;
ELSIF (nStatus AND 16#4F) = 16#40 THEN
	F_GetCoDS402State := E_CoDS402States.DS402STATE_SwitchOnDisabled;
ELSIF (nStatus AND 16#6F) = 16#21 THEN
	F_GetCoDS402State := E_CoDS402States.DS402STATE_ReadyToSwitchOn;
ELSIF (nStatus AND 16#6F) = 16#23 THEN
	F_GetCoDS402State := E_CoDS402States.DS402STATE_SwitchedOn;
ELSIF (nStatus AND 16#6F) = 16#27 THEN
	F_GetCoDS402State := E_CoDS402States.DS402STATE_OperationEnabled;
ELSIF (nStatus AND 16#6F) = 16#07 THEN
	F_GetCoDS402State := E_CoDS402States.DS402STATE_QuickStopActive;
ELSIF (nStatus AND 16#1400) = 16#1400 THEN
	F_GetCoDS402State := E_CoDS402States.DS402STATE_HomingCompleted;
ELSIF (nStatus AND 16#4F) = 16#0F THEN
	F_GetCoDS402State := E_CoDS402States.DS402STATE_FaultReactionActive;
ELSIF (nStatus AND 16#4F) = 16#08 THEN
	F_GetCoDS402State := E_CoDS402States.DS402STATE_Fault;
ELSE
	F_GetCoDS402State := E_CoDS402States.DS402STATE_Notspecified;
END_IF

END_FUNCTION

// ---- MainProgs/PC_Control.TcPOU
PROGRAM PC_Control
VAR
	fbWriteInd  	: ADSWRITEIND;
	fbWriteRes  	: ADSWRITERES;
	fbReadInd		: ADSREADIND;
	fbReadRes		: ADSREADRES;
	fbReadWriteInd	: ADSRDWRTIND;
	fbReadWriteRes	: ADSRDWRTRES;
	
	fbGetObjPropChecksum : FB_GetObjPropChecksum;
	
	uData			: U_AdsData;
	
	aBytes			: ARRAY[0..5] OF BYTE;
	nReadDataUSINT	: USINT;
	nDataUSINT		: USINT;	
 	nDataUINT		: UINT;
	nDataDINT		: DINT;
	nDataINT		: INT;
	stHardwareId	: ST_HardwareId;
	nObjectId		: UINT;
	stError			: ST_Error;
	stStepStatus	: ST_StepStatus;
	pMzTool			: POINTER TO FB_MzBase;
	pSequence		: POINTER TO FB_Sequence;
	pObject			: POINTER TO FB_Object;
	
	//Variablen für A_ExeAction
	eAction			: E_Action;
	
	stHardwareInfo	: ST_HardwareInfo;
	stPlcInfo		: ST_PlcInfo;
	aActiveActions	: ARRAY[0..9] OF ST_ActionStatus;
	
END_VAR

VAR CONSTANT
        READ_OBJECT_CHECKSUM	: UDINT := 16#80000002;
        READ_CONFIG_CHECKSUM	: UDINT := 16#80000003;
        ACTIVATE_CONFIG 		: UDINT := 16#80000004;
        READ_ACTIVATE_STATE 	: UDINT := 16#80000005;
        DELETE_ALL_OBJECTS 		: UDINT := 16#80000006;
        DELETE_OBJECT 			: UDINT := 16#80000007;
        CREATE_OBJECT 			: UDINT := 16#80000008;
        WRITE_ALL_PROPS 		: UDINT := 16#80000009;
        WRITE_SINGLE_PROP 		: UDINT := 16#8000000A;
        READ_ALL_PROPS 			: UDINT := 16#8000000B;
		READ_OBJECT_IDS 		: UDINT := 16#8000000D;
        UPLOAD_SEQU_STEP 		: UDINT := 16#80000011;
        UPLOAD_SEQU_CONDI 		: UDINT := 16#80000012;
        DELETE_SEQUENCE 		: UDINT := 16#80000013;
        CHANGE_MODE 			: UDINT := 16#80000018;
        RESET_ERROR 			: UDINT := 16#80000019;
        WRITE_HW_PROP 			: UDINT := 16#8000001A;
        READ_HW_PROP 			: UDINT := 16#8000001B;
        INTERACT_RESPONSE 		: UDINT := 16#8000001C;
        SETUP_AXIS 				: UDINT := 16#8000001D;
        FIRMWARE_UPDATE_CAN 	: UDINT := 16#8000001E;
		READ_ERROR				: UDINT := 16#8000001F;
		CREATE_SEQUENCE			: UDINT := 16#80000020;
		STOP					: UDINT := 16#80000021;
		GET_MODIFIED_OBJECT		: UDINT := 16#80000022;
		READ_HW_INFO			: UDINT := 16#80000023;
		READ_PLC_INFO			: UDINT := 16#80000024;
		INTERLOCK				: UDINT := 16#80000025;
		SAVE_CURR_CONFIG		: UDINT := 16#80000026;
		DELETE_CURR_CONFIG		: UDINT := 16#80000027;
		READ_MINMAXACT_POS		: UDINT := 16#80000028;
		RESET_PLC				: UDINT := 16#80000029;
        EXECUTE_ACTION 			: UDINT := 16#800000F0;
		STOP_ACTION 			: UDINT := 16#800000F1;
		PAUSE_ACTION 			: UDINT := 16#800000F2;
		CONTINUE_ACTION			: UDINT := 16#800000F3;
		READ_ACTIVE_ACTIONS		: UDINT := 16#800000F4;
END_VAR

fbWriteRes(RESPOND:= FALSE );(* Reset response function block *)
fbWriteInd(CLEAR:= FALSE );(* Trigger indication function block *)
fbReadRES(RESPOND:= FALSE );(* Reset response function block *)
fbReadInd(CLEAR:= FALSE );(* Trigger indication function block *)
fbReadWriteRes(RESPOND:= FALSE );(* Reset response function block *)
fbReadWriteInd(CLEAR:= FALSE );(* Trigger indication function block *)

IF fbWriteInd.VALID THEN
	fbWriteRes.RESULT := 0;
	CASE fbWriteInd.IDXGRP OF
		ACTIVATE_CONFIG:	//ActivateConfig
			fbWriteRes.RESULT := MainDispacher.M_ActivateConfig();
		SAVE_CURR_CONFIG:	//Aktuelle Konfiguration speichern - wird beim Plc-Neustart wieder geladen
			fbWriteRes.RESULT := MainDispacher.M_SaveConfig();
		DELETE_CURR_CONFIG:	//Gespeicherte Konfiguration löschen
			fbWriteRes.RESULT := MainDispacher.M_DeleteConfig();
		DELETE_ALL_OBJECTS:	//DeleteAllObjects
			//Länge überprüfen
			IF fbWriteInd.LENGTH = 0 THEN
				IF MainDispacher.eCurrentMode = E_MachineMode.MACHINEMODE_Config THEN //im Config-Modus?
					fbWriteRes.RESULT := fbObjectDirectory.M_DeleteAllObj();
				ELSE
					fbWriteRes.RESULT := E_ErrorIdCmd.ERRORID_WrongMode;	//Error: nicht im Config-Modus
				END_IF
			ELSE
				fbWriteRes.RESULT := DEVICE_INVALIDSIZE;
			END_IF
		DELETE_OBJECT:
			IF fbWriteInd.LENGTH = 0 THEN
				IF MainDispacher.eCurrentMode = E_MachineMode.MACHINEMODE_Config THEN //im Config-Modus?
					IF MainDispacher.eCurrentState = E_MachineState.MACHINESTATE_Idle THEN
						fbWriteRes.RESULT := fbObjectDirectory.M_DeleteObject(UDINT_TO_UINT(fbWriteInd.IDXOFFS));
					ELSE
						fbWriteRes.RESULT := E_ErrorIdCmd.ERRORID_InvalidState; //Error: nicht in Idle
					END_IF
				ELSE
					fbWriteRes.RESULT := E_ErrorIdCmd.ERRORID_WrongMode; //Error: nicht im Config-Modus
				END_IF
			ELSE
				fbWriteRes.RESULT := DEVICE_INVALIDSIZE;
			END_IF
		WRITE_ALL_PROPS: //WriteAllProps
			//Länge überprüfen
			IF fbWriteInd.LENGTH > 0 AND fbWriteInd.LENGTH <= SIZEOF(uData.stCmdData) THEN
				IF MainDispacher.eCurrentMode = E_MachineMode.MACHINEMODE_Config THEN //im Config-Modus?
					MEMSET(ADR(uData.stCmdData),0,SIZEOF(uData.stCmdData));
					MEMCPY(ADR(uData.stCmdData),fbWriteInd.DATAADDR,fbWriteInd.LENGTH);
					//Existiert Object?
					nObjectId := uData.stCmdData.aHeader[0];
					pObject := fbObjectDirectory.M_GetObjPointer(nObjectId);
					IF pObject > 0 THEN
						fbWriteRes.RESULT := pObject^.M_SetAllProps(uData.stCmdData);
					ELSE
						fbWriteRes.RESULT := E_ErrorIdCmd.ERRORID_ObjectNotExists;	//Error: Object existiert nicht
					END_IF
				ELSE
					fbWriteRes.RESULT := E_ErrorIdCmd.ERRORID_WrongMode;	//Error: nicht im Config-Modus
				END_IF
			ELSE
				fbWriteRes.RESULT := DEVICE_INVALIDSIZE;
			END_IF
		WRITE_SINGLE_PROP:	//WriteSingleProp
			//Länge überprüfen
			IF fbWriteInd.LENGTH > 0 AND fbWriteInd.LENGTH <= SIZEOF(uData.stCmdData) THEN
				MEMSET(ADR(uData.stCmdData),0,SIZEOF(uData.stCmdData));
				MEMCPY(ADR(uData.stCmdData),fbWriteInd.DATAADDR,fbWriteInd.LENGTH);
				//Existiert Object?
				nObjectId := uData.stCmdData.aHeader[0];
				pObject := fbObjectDirectory.M_GetObjPointer(nObjectId);
				IF pObject > 0 THEN
					fbWriteRes.RESULT := pObject^.M_SetSingleProp(uData.stCmdData);
				ELSE
					fbWriteRes.RESULT := E_ErrorIdCmd.ERRORID_ObjectNotExists;	//Error: Object existiert nicht
				END_IF
			ELSE
				fbWriteRes.RESULT := DEVICE_INVALIDSIZE;
			END_IF
		CREATE_SEQUENCE:	//Neue Sequence erstellen
			//Länge überprüfen
			IF fbWriteInd.LENGTH = 2 THEN
				IF MainDispacher.P_eCurrentState = E_MachineState.MACHINESTATE_Idle THEN
					MEMCPY(ADR(nDataUINT),fbWriteInd.DATAADDR,fbWriteInd.LENGTH);
					IF NOT fbSequenceList.M_Add(fbWriteInd.IDXOFFS,nDataUINT) THEN
						RETURN;
					END_IF
				ELSE
					fbWriteRes.RESULT := E_ErrorIdCmd.ERRORID_InvalidState;
				END_IF
			ELSE
				fbWriteRes.RESULT := DEVICE_INVALIDSIZE;
			END_IF
		UPLOAD_SEQU_STEP:	//Upload SequenceStep
			//Länge überprüfen
			IF fbWriteInd.LENGTH >= 32 AND fbWriteInd.LENGTH <= SIZEOF(uData.stCmdData) THEN
				IF MainDispacher.P_eCurrentState = E_MachineState.MACHINESTATE_Idle THEN
					MEMSET(ADR(uData.stCmdData),0,SIZEOF(uData.stCmdData));
					MEMCPY(ADR(uData.stCmdData),fbWriteInd.DATAADDR,fbWriteInd.LENGTH);
					pSequence := fbSequenceList.M_Get(fbWriteInd.IDXOFFS);
					IF pSequence > 0 THEN
						fbWriteRes.RESULT := pSequence^.M_AddStep(uData.stCmdData);
					ELSE
						fbWriteRes.RESULT := E_ErrorIdCmd.ERRORID_SequenceNotExists;
					END_IF
				ELSE
					fbWriteRes.RESULT := E_ErrorIdCmd.ERRORID_InvalidState;
				END_IF
			ELSE
				fbWriteRes.RESULT := DEVICE_INVALIDSIZE;
			END_IF
		UPLOAD_SEQU_CONDI:	//Upload SequenceCondi
			//Länge überprüfen
			IF fbWriteInd.LENGTH = 24 THEN
				MEMSET(ADR(uData.stCmdData),0,SIZEOF(uData.stCmdData));
				MEMCPY(ADR(uData.stCmdData),fbWriteInd.DATAADDR,fbWriteInd.LENGTH);
				IF MainDispacher.P_eCurrentState = E_MachineState.MACHINESTATE_Idle THEN
					pSequence := fbSequenceList.M_Get(fbWriteInd.IDXOFFS);
					IF pSequence > 0 THEN
						fbWriteRes.RESULT := pSequence^.M_AddCondi(uData.stCmdData);
					ELSE
						fbWriteRes.RESULT := E_ErrorIdCmd.ERRORID_SequenceNotExists;
					END_IF
				ELSE
					fbWriteRes.RESULT := E_ErrorIdCmd.ERRORID_InvalidState;
				END_IF
			ELSE
				fbWriteRes.RESULT := DEVICE_INVALIDSIZE;
			END_IF
		DELETE_SEQUENCE: //Alle Sequenzen löschen
			IF MainDispacher.eCurrentState = E_MachineState.MACHINESTATE_Idle THEN
				fbWriteRes.RESULT := 0;
				//Alle Sequencen löschen
				IF NOT fbSequenceList.M_Delete() THEN
					fbWriteRes.RESULT := 1;
				END_IF
			ELSE
				fbWriteRes.RESULT := E_ErrorIdCmd.ERRORID_InvalidState;
			END_IF
 		CHANGE_MODE: //Change Mode
			//Länge überprüfen
			IF fbWriteInd.LENGTH = 0 THEN
				fbWriteRes.RESULT := MainDispacher.M_ChangeMode(UDINT_TO_USINT(fbWriteInd.IDXOFFS));
			ELSE
				fbWriteRes.RESULT := DEVICE_INVALIDSIZE;
			END_IF
		RESET_ERROR:
			//Länge überprüfen
			IF fbWriteInd.LENGTH = 0 THEN
				MainDispacher.M_ResetError();
			ELSE
				fbWriteRes.RESULT := DEVICE_INVALIDSIZE;
			END_IF
		WRITE_HW_PROP:	//HardwareProp schreiben
			//Länge überprüfen
			IF fbWriteInd.LENGTH = 10 THEN
				IF MainDispacher.eCurrentMode = E_MachineMode.MACHINEMODE_Config OR 
					MainDispacher.eCurrentMode = E_MachineMode.MACHINEMODE_Maintenance THEN
					MEMCPY(ADR(stHardwareId),fbWriteInd.DATAADDR, 3);
					MEMCPY(ADR(nDataUINT), fbWriteInd.DATAADDR + 4, 2);
					MEMCPY(ADR(nDataDINT), fbWriteInd.DATAADDR + 6, 4);
					fbWriteRes.RESULT := fbSettings.M_WriteProp(stHardwareId:= stHardwareId,ePropType:= nDataUINT,nValue:= nDataDINT); 
				ELSE
					fbWriteRes.RESULT := E_ErrorIdCmd.ERRORID_WrongMode;	//Error: nicht im Config bzw. Maintenance-Mode
				END_IF
			ELSE
				fbWriteRes.RESULT := DEVICE_INVALIDSIZE;
			END_IF
		INTERACT_RESPONSE:	//Antwort auf einen InterRequest
			//Länge überprüfen
			IF fbWriteInd.LENGTH = 24 THEN
				MEMSET(ADR(uData.stCmdData),0,SIZEOF(uData.stCmdData));
				MEMCPY(ADR(uData.stCmdData),fbWriteInd.DATAADDR,fbWriteInd.LENGTH);
				stInterResponse.nObjectId := uData.stCmdData.aHeader[0];
				stInterResponse.eInteractMessageType := uData.stCmdData.aHeader[1];
				stInterResponse.nArg1 := uData.stCmdData.n32Data[0];
				stInterResponse.nArg2 := uData.stCmdData.n32Data[1];
				stInterResponse.nArg3 := uData.stCmdData.n32Data[2];
				stInterResponse.nArg4 := uData.stCmdData.n32Data[3];
			ELSE
				fbWriteRes.RESULT := DEVICE_INVALIDSIZE;
			END_IF
		SETUP_AXIS:
			//Länge überprüfen
			IF fbWriteInd.LENGTH = 24 THEN
				MEMSET(ADR(uData.stCmdData),0,SIZEOF(uData.stCmdData));
				MEMCPY(ADR(uData.stCmdData.n32Data) ,fbWriteInd.DATAADDR,fbWriteInd.LENGTH);
				fbWriteRes.RESULT := MainDispacher.M_SetupAxis(uData.stCmdData);
			ELSE
				fbWriteRes.RESULT := DEVICE_INVALIDSIZE;
			END_IF
		STOP:
			MainDispacher.M_StopAll();
			
		STOP_ACTION:
			IF fbWriteInd.LENGTH = 0 THEN
				fbWriteRes.RESULT := MainDispacher.M_StopAction(UDINT_TO_UINT(fbWriteInd.IDXOFFS));
			ELSE
				fbWriteRes.RESULT := DEVICE_INVALIDSIZE;
			END_IF
		PAUSE_ACTION:
			IF fbWriteInd.LENGTH = 0 THEN
				fbWriteRes.RESULT := MainDispacher.M_PauseAction(UDINT_TO_UINT(fbWriteInd.IDXOFFS));
			ELSE
				fbWriteRes.RESULT := DEVICE_INVALIDSIZE;
			END_IF
		CONTINUE_ACTION:
			IF fbWriteInd.LENGTH = 0 THEN
				fbWriteRes.RESULT := MainDispacher.M_ContinueAction(UDINT_TO_UINT(fbWriteInd.IDXOFFS));
			ELSE
				fbWriteRes.RESULT := DEVICE_INVALIDSIZE;
			END_IF
		INTERLOCK:
			//Länge überprüfen
			IF fbWriteInd.LENGTH = 1 THEN
				MEMCPY(ADR(nDataUSINT),fbWriteInd.DATAADDR,fbWriteInd.LENGTH);
				IF fbWriteInd.IDXOFFS = 0 OR fbWriteInd.IDXOFFS = 1 THEN
					fbWriteRes.RESULT := pFbSafety^.M_Control(nDataUSINT);
				ELSIF fbWriteInd.IDXOFFS = 2 THEN
					{IF defined(variable: fbSafetyStacker)}
					fbWriteRes.RESULT := fbSafetyStacker.M_Control(nDataUSINT);
					{ELSE}
					fbWriteRes.RESULT := DEVICE_INVALIDOFFSET;
					{END_IF}
				ELSE
					fbWriteRes.RESULT := DEVICE_INVALIDOFFSET;
				END_IF
			ELSE
				fbWriteRes.RESULT := DEVICE_INVALIDSIZE;
			END_IF
		FIRMWARE_UPDATE_CAN:
			IF fbWriteInd.LENGTH = 0 THEN
				fbWriteRes.RESULT := MainDispacher.M_DeviceFirmwUpdate(UDINT_TO_USINT(fbWriteInd.IDXOFFS));
			ELSE
				fbWriteRes.RESULT := DEVICE_INVALIDSIZE;
			END_IF
		RESET_PLC:
			IF fbWriteInd.LENGTH = 0 THEN
				fbWriteRes.RESULT := MainDispacher.M_ResetPlc();
			ELSE
				fbWriteRes.RESULT := DEVICE_INVALIDSIZE;
			END_IF
	ELSE //Ads-Error InvalidIndexOffset
		fbWriteRes.RESULT := DEVICE_INVALIDGRP;
	END_CASE
	fbWriteRes(NETID:= fbWriteInd.NETID,PORT:= fbWriteInd.PORT, INVOKEID:= fbWriteInd.INVOKEID, RESPOND:= TRUE);
	fbWriteInd(CLEAR := TRUE);
ELSIF fbReadInd.VALID THEN
	fbReadRES.RESULT := NOERR;
	CASE fbReadInd.IDXGRP OF
		READ_OBJECT_CHECKSUM:	//ReadObjectCheckSum	
			//Länge überprüfen
			IF fbReadInd.LENGTH = 2 THEN
				//Checksum aller Properties aller Objecte ermitteln
				fbGetObjPropChecksum(bExecute:= TRUE, ObjectDirectoryRef:= fbObjectDirectory);
				IF fbGetObjPropChecksum.bBusy THEN
					RETURN;
				ELSE
					nDataUINT := fbGetObjPropChecksum.nResult;
					fbGetObjPropChecksum(bExecute:= FALSE, ObjectDirectoryRef:= fbObjectDirectory);
				END_IF
				fbReadRES.DATAADDR := ADR(nDataUINT);
			ELSE
				fbReadRES.RESULT := DEVICE_INVALIDSIZE;
			END_IF
		READ_CONFIG_CHECKSUM:	//ReadConfigCheckSum
			//Länge überprüfen
			IF fbReadInd.LENGTH = 2 THEN
				nDataUINT := fbObjectDirectory.M_GetConfigCheckSum();	
				fbReadRES.DATAADDR := ADR(nDataUINT);
			ELSE
				fbReadRES.RESULT := DEVICE_INVALIDSIZE;
			END_IF
		READ_ACTIVATE_STATE:	//Read AktivateState
			//Länge überprüfen
			IF fbReadInd.LENGTH = 1 THEN
				nReadDataUSINT := BOOL_TO_USINT(fbConfiguration.P_bActivated);
				fbReadRES.DATAADDR := ADR(nReadDataUSINT);
			ELSE
				fbReadRES.RESULT := DEVICE_INVALIDSIZE;
			END_IF
		READ_ALL_PROPS:	//ReadAllProps
			//Länge überprüfen
			IF fbReadInd.LENGTH > 0  AND fbReadInd.LENGTH <= SIZEOF(uData.stCmdData) THEN
				MEMSET(ADR(uData.stCmdData),0,SIZEOF(uData.stCmdData));
				nObjectId := UDINT_TO_UINT(fbReadInd.IDXOFFS);
				pObject := fbObjectDirectory.M_GetObjPointer(nObjectId);
				IF pObject > 0 THEN
					fbReadRES.RESULT :=  pObject^.M_GetAllProps(uData.stCmdData);
					//Crc bilden und in Header[3] schreiben
					
					uData.stCmdData.aHeader[3] := F_DATA_TO_CRC16_CCITT(ADR(uData.stCmdData.n32Data[0]),pObject^.P_nNoOfProps * 4,16#FFFF);
				ELSE
					fbReadRES.RESULT := E_ErrorIdCmd.ERRORID_ObjectNotExists;	//Error: Object existiert nicht
				END_IF
				IF fbObjectDirectory.M_GetObjType(nObjectId) <> E_ObjectType.OBJECTTYPE_UNDEFINED THEN
					fbReadRES.RESULT :=  fbObjectDirectory.M_GetObjPointer(nObjectId)^.M_GetAllProps(uData.stCmdData);
					//Crc bilden und in Header[3] schreiben
					uData.stCmdData.aHeader[3] := F_DATA_TO_CRC16_CCITT(ADR(uData.stCmdData.n32Data[0]),fbObjectDirectory.M_GetObjPointer(nObjectId)^.P_nNoOfProps * 4,16#FFFF);
					fbReadRES.DATAADDR := ADR(uData.stCmdData);
				ELSE
					fbReadRES.RESULT := E_ErrorIdCmd.ERRORID_ObjectNotExists;	//Error: Object existiert nicht
				END_IF
			ELSE
				fbReadRES.RESULT := DEVICE_INVALIDSIZE;
			END_IF
		GET_MODIFIED_OBJECT:
			//Länge überprüfen
			MEMSET(ADR(uData.stCmdData),0,SIZEOF(uData.stCmdData));
			IF fbReadInd.LENGTH = 2 THEN
				//nächtses Object aus List holen
				nObjectId := fbObjectDirectory.M_GetChangedObjId();
				IF nObjectId > 0 THEN
					fbObjectDirectory.M_RemoveObjChange(nObjectId);
					nDataUINT := nObjectId;
				ELSE
					nDataUINT := 0;
				END_IF
				fbReadRES.DATAADDR := ADR(nDataUINT);
			ELSE
				fbReadRES.RESULT := DEVICE_INVALIDSIZE;
			END_IF
		READ_HW_INFO:
			//Länge überprüfen
			IF fbReadInd.LENGTH = 44 THEN
				IF fbReadInd.IDXOFFS = 0 THEN
					HwInfoList.M_ResetPointer();
				END_IF
				stHardwareInfo := HwInfoList.M_GetNext();
				fbReadRES.DATAADDR := ADR(stHardwareInfo);
			ELSE
				fbReadRES.RESULT := DEVICE_INVALIDSIZE;
			END_IF
		READ_PLC_INFO:
			//Länge überprüfen
			IF fbReadInd.LENGTH = SIZEOF(stPlcInfo) THEN
				stPlcInfo := GVL_Hardware.stPlcInfo;
				fbReadRES.DATAADDR := ADR(stPlcInfo);
			ELSE
				fbReadRES.RESULT := DEVICE_INVALIDSIZE;
			END_IF
		READ_MINMAXACT_POS:
			//Länge überprüfen
			IF fbReadInd.LENGTH <= 36 THEN
				//Checken, ob Object ein MzTool
				nObjectId := UDINT_TO_UINT(fbReadInd.IDXOFFS);
				IF fbObjectDirectory.M_ObjIsMzTool(nObjectId) THEN
					pMzTool := fbObjectDirectory.M_GetObjPointer(nObjectId);
					pMzTool^.M_GetMinMaxActPos(ADR(uData.aDINT_20));
					fbReadRES.DATAADDR := ADR(uData.aDINT_20);
				ELSE
					fbReadRES.RESULT := E_ErrorIdObjMgmt.ERRORID_IsNoMzTool;
				END_IF
			ELSE
				fbReadRES.RESULT := DEVICE_INVALIDSIZE;
			END_IF
		READ_ACTIVE_ACTIONS:
			//Länge überprüfen
			IF fbReadInd.LENGTH = 90 THEN
				ActionDispacher.M_GetActionInfoArray(ADR(aActiveActions));
				fbReadRES.DATAADDR := ADR(aActiveActions);
			ELSE
				fbReadRES.RESULT := DEVICE_INVALIDSIZE;
			END_IF
		READ_OBJECT_IDS:
			//Länge überprüfen (muss genau Anzahl Objekte * 2 sein)
			IF fbReadInd.LENGTH = fbObjectDirectory.nCntObject * 2 THEN
				//Die ObjectIDs stehen nacheinander in einem ARRAY[0..n] OF UINT
				fbReadRES.RESULT := fbObjectDirectory.M_GetObjIdStream(uData.aUINT_1000);
				fbReadRES.DATAADDR := ADR(uData);
			ELSE
				fbReadRES.RESULT := DEVICE_INVALIDSIZE;
			END_IF
	ELSE //Ads-Error InvalidIndexOffset
		fbReadRES.RESULT := DEVICE_INVALIDGRP;
	END_CASE
	fbReadRes(NETID:= fbReadInd.NETID, PORT:= fbReadInd.PORT, INVOKEID:= fbReadInd.INVOKEID, LEN:= fbReadInd.LENGTH, RESPOND:= TRUE); 
	fbReadInd(CLEAR := TRUE ); 
ELSIF fbReadWriteInd.VALID THEN
	CASE fbReadWriteInd.IDXGRP OF
		CREATE_OBJECT:	//CreateObject
			//Längen überprüfen
			IF fbReadWriteInd.WRTLENGTH <= (SIZEOF(uData.stCmdData) + 2) AND fbReadWriteInd.RDLENGTH = 6 THEN
				IF MainDispacher.eCurrentMode = E_MachineMode.MACHINEMODE_Config THEN //im Config-Modus?
					MEMCPY(ADR(nDataINT),fbReadWriteInd.DATAADDR,2); //Index
					MEMSET(ADR(uData.stCmdData),0,SIZEOF(uData.stCmdData));
					MEMCPY(ADR(uData.stCmdData),fbReadWriteInd.DATAADDR + 2,fbReadWriteInd.WRTLENGTH);
					fbReadWriteRes.RESULT := fbObjectDirectory.M_CreateObject(nDataINT, refCmdData:= uData.stCmdData,nNotifyId=>nDataDINT);
					MEMCPY(ADR(aBytes),ADR(nDataDINT),4); //NotifyId zurückgeben
					MEMCPY(ADR(aBytes)+4,ADR(uData.stCmdData.aHeader[0]),2); //ObjectId zurückgeben
					fbReadWriteRes.DATAADDR := ADR(aBytes); 
				ELSE
					fbReadWriteRes.RESULT := E_ErrorIdCmd.ERRORID_WrongMode; //Error: nicht im Config-Modus
				END_IF				
			ELSE
				fbReadWriteRes.RESULT := DEVICE_INVALIDSIZE;
			END_IF
		READ_HW_PROP:	//Read HardwareProp
			//Längen überprüfen
			IF fbReadWriteInd.WRTLENGTH = 6 AND fbReadWriteInd.RDLENGTH = 4 THEN
				MEMCPY(ADR(stHardwareId),fbReadWriteInd.DATAADDR,3);
				MEMCPY(ADR(nDataUINT),fbReadWriteInd.DATAADDR + 4,2);
				fbReadWriteRes.RESULT := fbSettings.M_ReadProp(stHardwareId:= stHardwareId, ePropType:= nDataUINT,nValue=> nDataDINT);
				fbReadWriteRes.DATAADDR := ADR(nDataDINT);
			ELSE
				fbReadWriteRes.RESULT := DEVICE_INVALIDSIZE;
			END_IF
		EXECUTE_ACTION:	//ExecuteAction
			//Länge überprüfen
			IF fbReadWriteInd.WRTLENGTH <= 160 AND fbReadWriteInd.RDLENGTH = 2 THEN
				eAction := UDINT_TO_UINT(fbReadWriteInd.IDXOFFS);
				MEMSET(ADR(uData.aDINT_40),0,SIZEOF(uData.aDINT_40));
				MEMCPY(ADR(uData.aDINT_40),fbReadWriteInd.DATAADDR,fbReadWriteInd.WRTLENGTH);
				stError := MainDispacher.M_ExeAction(eAction:= eAction, uData.aDINT_40,nActionId=>nDataUINT);
				fbReadWriteRes.DATAADDR := ADR(nDataUINT);
				fbReadWriteRes.RESULT := stError.ErrorId;
			ELSE
				fbWriteRes.RESULT := DEVICE_INVALIDSIZE;
			END_IF			
	ELSE //Ads-Error InvalidIndexOffset
		fbReadWriteRes.RESULT := DEVICE_INVALIDGRP;
	END_CASE
	fbReadWriteRes(NETID:= fbReadWriteInd.NETID, PORT:= fbReadWriteInd.PORT, INVOKEID:= fbReadWriteInd.INVOKEID, LEN:= fbReadWriteInd.RDLENGTH, RESPOND:= TRUE);
	fbReadWriteInd(CLEAR:= TRUE );
END_IF

END_PROGRAM

// ---- Configuration/FB_GetObjPropChecksum.TcPOU
FUNCTION_BLOCK FB_GetObjPropChecksum
VAR_INPUT
	bExecute : BOOL;
END_VAR
VAR_OUTPUT
	bBusy : BOOL;
	nResult : UINT;
END_VAR
VAR
	rTrig			: R_TRIG;
	nCounter		: USINT;
	wPrevChecksum	: WORD;
	nObjChecksum 	: UINT;
	iter			: FB_ObjCollectIteratorDeep;
END_VAR
VAR_IN_OUT
	ObjectDirectoryRef : FB_ObjectDirectory;
END_VAR

rTrig(CLK:= bExecute);
IF rTrig.Q THEN
	bBusy := TRUE;
	wPrevChecksum := 16#FFFF;
	ObjectDirectoryRef.objectList.M_GetIterator(iter);
END_IF

IF bExecute THEN
	nCounter := 0;
	WHILE iter.pNode > 0 AND_THEN iter.pNode^.P_pObject > 0 DO
		nObjChecksum := iter.pNode^.P_pObject^.M_GetPropCheckSum();
		wPrevChecksum := F_DATA_TO_CRC16_CCITT(ADR(nObjChecksum),SIZEOF(nObjChecksum),wPrevChecksum);
		nCounter := nCounter + 1;
		iter.M_Increment();
		IF nCounter = 100 THEN
			RETURN;
		END_IF
	END_WHILE
	nResult := wPrevChecksum;
	bBusy := FALSE;
ELSE
	bBusy := FALSE;
	nResult := 0;
END_IF

END_FUNCTION_BLOCK

// ---- Configuration/FB_ObjectDirectory.TcPOU
FUNCTION_BLOCK FB_ObjectDirectory

VAR_OUTPUT
	bIsInitialized			: BOOL;

	//Anzahl der jeweiligen Objekttypen, welche ins Objektverzeichnis eingetragen sind (Objektzählervariablen)
	nCntCamera				:UINT;
	nCntCartDispenser		:UINT;
	nCntCartDispStirrer		:UINT;
	nCntCartHolder			:UINT;
	nCntCustomUnitType1		:UINT;
	nCntCustomUnitType2		:UINT;
	nCntMultiCartHolder		:UINT;
	nCntHybridDispenser		:UINT;
	nCntDeloDot				:UINT;
	nCntDiluter				:UINT;
	nCntDiluter3Inputs		:UINT;
	nCntDrayPad				:UINT;
	nCntDummyTool			:UINT;
	nCntExposure			:UINT;
	nCntExtruder			:UINT;
	nCntFlipTubeHandler		:UINT;
	nCntFlipTubeRack		:UINT;
	nCntGripper				:UINT;
	nCntHighVoltTray		:UINT;
	nCntInkStation			:UINT;
	nCntLiquidReserve		:UINT;
	nCntLuer				:UINT;
	nCntMtpHolder			:UINT;
	nCntMZHead				:UINT;
	nCntNeedleRack			:UINT;
	nCntPassivPip			:UINT;
	nCntpHElectrode			:UINT;
	nCntpHElectrodeCapRack	:UINT;
	nCntPickPlacePip		:UINT;
	nCntPiezoPip			:UINT;
	nCntPortRack			:UINT;
	nCntPowderPip			:UINT;
	nCntPowderStation		:UINT;
	nCntReactor				:UINT;
	nCntSampleScan			:UINT;
	nCntSeptumRack			:UINT;
	nCntSeptumWaste			:UINT;
	nCntSinglePiezoHolder	:UINT;
	nCntStacker				:UINT;
	nCntSolenoidPip			:UINT;
	nCntStampMagazine		:UINT;
	nCntStampSupport		:UINT;
	nCntStroboscope			:UINT;
	nCntSubstHolder			:UINT;
	nCntSubstHolderUnistat	:UINT;
	nCntTipCalibrator		:UINT;
	nCntTipCleaner			:UINT;
	nCntTipCleanerGen2		:UINT;
	nCntTipRack				:UINT;
	nCntTitrationTool		:UINT;
	nCntTrayTransporter		:UINT;
	nCntTriplePip			:UINT;
	nCntTwinExtruder		:UINT;
	nCntTwinPiezoHolder		:UINT;
	nCntVacuumHandler		:UINT;
	nCntVermesDisp			:UINT;
	nCntVialRack			:UINT;
	nCntWashStation			:UINT;
	nCntWorkplate			:UINT;
	nCntWorkplateCamera		:UINT;
	nCntZLevelSensor		:UINT;
	
	//Anzahl der jeweiligeb Objecttypen, welche in InterfaceArrays eingetragen sind
	nCntObject			: UINT;
	
	//Anzahl der aktuellen benutzen NotificationIds
	nCntNotifiIds		: UINT;

END_VAR

VAR
	fbIdPool 			: FB_IdPool;
	a_pObjects 			: ARRAY[1..cMaxObjects] OF POINTER TO FB_Object;
	objectList			: FB_ObjCollection(0);
	deviceList			: FB_ObjCollection(0);	

	//Für ObjectChange
	fbList				: FB_LinkedListCtrl;
	hList				: T_HLINKEDLIST;
	nodes				: ARRAY [0..20] OF T_LinkedListEntry;
	
	//Notification MoveObject
	stObjectHasMoved	: ST_ObjHasMoved;
	
	pCartridge			: POINTER TO FB_Cartridge;	
	pFlipTube			: POINTER TO FB_FlipTube;	
	pMtp				: POINTER TO FB_Mtp;
	pNeedle				: POINTER TO FB_Needle;
	pNozzle				: POINTER TO FB_Nozzle;
	pPHElectrodeCap		: POINTER TO FB_pHElectrodeCap;		
	pPoint				: POINTER TO FB_Point;
	pPort				: POINTER TO FB_Port;
	pSeptum				: POINTER TO FB_Septum;
	pSlide				: POINTER TO FB_Slide;
	pSpotArray			: POINTER TO FB_SpotArray;	
	//pSpotPattern		: POINTER TO FB_SpotPattern;		
	pStamp				: POINTER TO FB_Stamp;
	pTip				: POINTER TO FB_Tip;
	pTray				: POINTER TO FB_TargetTray;
	pVial				: POINTER TO FB_Vial;
	pVialClosed			: POINTER TO FB_VialClosed;	
	//pWafer				: POINTER TO FB_Wafer;
	pCleaningBrush		: POINTER TO FB_CleaningBrush;
END_VAR

METHOD M_CheckCuboidCollision : BOOL
VAR_INPUT
	Cuboid : REFERENCE TO FB_Cuboid;
END_VAR

VAR
END_VAR
//Überprüft den übergebenen Quader darauf, dass er mit keinem Target auf der Workplate oder
//mit einem Tool in HomePos kollidiert. Punkte werden dabei ausgeschlossen.
//Das erste Problem besteht darin, dass ein Point in einem Target vertieft befinden kann (MTP)
//oder z.B. ein Punkt, der vermessen wurde und sich dadurch unterhalb des Targets befindet
//in diesem Fall muss genau dieses Target als Kollisionsobjekt ausgeschlossen werden
//also das Target, auf dem sich der Punkt befindet. Wie sieht es mit einem Slide aus? Wenn dieses 
//durch Vermessung etwas tiefer sitzt als sein Parent, dann macht das eigentlich nichts.

//Alle Targets durchlaufen? Mit einem Durchlauf? was ist, wenn es tausende Points gibt?
//afbWorkplate[1].
END_METHOD

METHOD  M_CreateObject : ERRORID
VAR_INPUT
	nIndex			: INT;	//Index in der ObjCollection ("-1" -> wird am Ende eingefügt)
	refCmdData		: REFERENCE TO ST_CmdData;
END_VAR
VAR_OUTPUT
	nNotifyId		: DINT;
END_VAR
VAR
	nObjectID		: UINT;
	eObjectType 	: E_ObjectType;
	nParentObjectId : UINT;
	pParentObject	: POINTER TO FB_Object;
	nParentSlotNr	: UINT;
	nNewIndex		: UINT;
END_VAR
//Methode zum Hinzufügen von Objecten ins Objektverzeichnis

nObjectID := fbIdPool.M_GetId();
IF nObjectID = 0 THEN
	M_CreateObject := E_ErrorIdObjMgmt.ERRORID_CntObjectsExceeded;	//Rückgabe Error
	RETURN;	
END_IF

eObjectType := refCmdData.aHeader[0];

IF (nObjectID  > 0) AND (nObjectID <= cMaxObjects) THEN
	IF a_pObjects[nObjectID] <> 0 THEN	//ObjectID schon vorhanden
		M_CreateObject := E_ErrorIdObjMgmt.ERRORID_ObjectIDAlreadyExists;
		RETURN;
	END_IF
ELSE
	M_CreateObject := E_ErrorIdObjMgmt.ERRORID_CntObjectsExceeded;	//Rückgabe Error
	RETURN;
END_IF

CASE eObjectType OF

	E_ObjectType.OBJECTTYPE_Camera:	//Camera, Mikroskop, Scanner o.ä.
		IF nCntCamera = cMaxCameras THEN	//maximale Anzahl des spez.Objecttypes erreicht, Object kann nicht angelegt werden
			M_CreateObject := E_ErrorIdObjMgmt.ERRORID_CntCamerasExceeded;	//Rückgabe Error
			RETURN;
		ELSE
			nCntCamera := nCntCamera + 1;
			a_pObjects[nObjectID] := ADR(afbCamera[nCntCamera]);
			afbCamera[nCntCamera].P_nObjectID := nObjectID;
			nCntNotifiIds := nCntNotifiIds + 1;
			afbCamera[nCntCamera].P_nNotifyId := nCntNotifiIds;
			nNotifyId := nCntNotifiIds;
 		END_IF

	E_ObjectType.OBJECTTYPE_Cartridge:	//Kartusche auf einem Rack
		pCartridge := __NEW(FB_Cartridge);
		pCartridge^.P_nObjectID := nObjectID;
		a_pObjects[nObjectID] := pCartridge;	
		
	E_ObjectType.OBJECTTYPE_CartDispenser:
		IF nCntCartDispenser = cMaxCartDisp THEN	//maximale Anzahl des spez.Objecttypes erreicht, Object kann nicht angelegt werden
			M_CreateObject := E_ErrorIdObjMgmt.ERRORID_CntCartridgeDispExceeded; //Rückgabe Error
			RETURN;
		ELSE
			nCntCartDispenser := nCntCartDispenser + 1;
			a_pObjects[nObjectID] := ADR(afbCartDisp[nCntCartDispenser]);
			afbCartDisp[nCntCartDispenser].P_nObjectID := nObjectID;
			nCntNotifiIds := nCntNotifiIds + 1;
			afbCartDisp[nCntCartDispenser].P_nNotifyId := nCntNotifiIds;
			nNotifyId := nCntNotifiIds;
 		END_IF
	E_ObjectType.OBJECTTYPE_CartDispStirrer:
		IF nCntCartDispStirrer = cMaxCartDispStirrer THEN	//maximale Anzahl des spez.Objecttypes erreicht, Object kann nicht angelegt werden
			M_CreateObject := E_ErrorIdObjMgmt.ERRORID_CntCartridgeDispStirrerExceeded; //Rückgabe Error
			RETURN;
		ELSE
			nCntCartDispStirrer := nCntCartDispStirrer + 1;
			a_pObjects[nObjectID] := ADR(afbCartDispStirrer[nCntCartDispStirrer]);
			afbCartDispStirrer[nCntCartDispStirrer].P_nObjectID := nObjectID;
			nCntNotifiIds := nCntNotifiIds + 1;
			afbCartDispStirrer[nCntCartDispStirrer].P_nNotifyId := nCntNotifiIds;
			nNotifyId := nCntNotifiIds;
 		END_IF
E_ObjectType.OBJECTTYPE_CartHolder:
		IF nCntCartHolder = cMaxCartHolder THEN	//maximale Anzahl des spez.Objecttypes erreicht, Object kann nicht angelegt werden
			M_CreateObject := E_ErrorIdObjMgmt.ERRORID_CntCartridgeHolderExceeded;	//Rückgabe Error
			RETURN;
		ELSE
			nCntCartHolder := nCntCartHolder + 1;
			a_pObjects[nObjectID] := ADR(afbCartHolder[nCntCartHolder]);
			afbCartHolder[nCntCartHolder].P_nObjectID := nObjectID;
			nCntNotifiIds := nCntNotifiIds + 1;
			afbCartHolder[nCntCartHolder].P_nNotifyId := nCntNotifiIds;
			nNotifyId := nCntNotifiIds;
 		END_IF
		
	E_ObjectType.OBJECTTYPE_CleaningBrush:
		pCleaningBrush := __NEW(FB_CleaningBrush);
		pCleaningBrush^.P_nObjectID := nObjectID;
		a_pObjects[nObjectID] := pCleaningBrush;	
		
	E_ObjectType.OBJECTTYPE_CustomUnitType1:
		IF nCntCustomUnitType1 = cMaxCustomUnitTyp1 THEN //maximale Anzahl des spez.Objecttypes erreicht, Object kann nicht angelegt werden
			M_CreateObject := E_ErrorIdObjMgmt.ERRORID_CntCustomUnitType1Exceeded; //Rückgabe Error
			RETURN;
		ELSE
			nCntCustomUnitType1 := nCntCustomUnitType1 + 1;
			a_pObjects[nObjectID] := ADR(afbCustomUnitType1[nCntCustomUnitType1]);
			afbCustomUnitType1[nCntCustomUnitType1].P_nObjectID := nObjectID;
			nCntNotifiIds := nCntNotifiIds + 1;
			afbCustomUnitType1[nCntCustomUnitType1].P_nNotifyId := nCntNotifiIds;			
			nNotifyId := nCntNotifiIds;
		END_IF
		
	E_ObjectType.OBJECTTYPE_CustomUnitType2:
		IF nCntCustomUnitType2 = cMaxCustomUnitTyp2 THEN //maximale Anzahl des spez.Objecttypes erreicht, Object kann nicht angelegt werden
			M_CreateObject := E_ErrorIdObjMgmt.ERRORID_CntCustomUnitType2Exceeded; //Rückgabe Error
			RETURN;
		ELSE
			nCntCustomUnitType2 := nCntCustomUnitType2 + 1;
			a_pObjects[nObjectID] := ADR(afbCustomUnitType2[nCntCustomUnitType2]);
			afbCustomUnitType2[nCntCustomUnitType2].P_nObjectID := nObjectID;
			nCntNotifiIds := nCntNotifiIds + 1;
			afbCustomUnitType2[nCntCustomUnitType2].P_nNotifyId := nCntNotifiIds;			
			nNotifyId := nCntNotifiIds;
		END_IF

	E_ObjectType.OBJECTTYPE_MultiCartHolder:
		IF nCntMultiCartHolder = cMaxMultiCartHolder THEN	//maximale Anzahl des spez.Objecttypes erreicht, Object kann nicht angelegt werden
			M_CreateObject := E_ErrorIdObjMgmt.ERRORID_CntMultiCartridgeHolderExceeded;	//Rückgabe Error
			RETURN;
		ELSE
			nCntMultiCartHolder := nCntMultiCartHolder + 1;
			a_pObjects[nObjectID] := ADR(afbMultiCartHolder[nCntMultiCartHolder]);
			afbMultiCartHolder[nCntMultiCartHolder].P_nObjectID := nObjectID;
			nCntNotifiIds := nCntNotifiIds + 1;
			afbMultiCartHolder[nCntMultiCartHolder].P_nNotifyId := nCntNotifiIds;
			nNotifyId := nCntNotifiIds;
		END_IF
		
	E_ObjectType.OBJECTTYPE_HybridDispenser:
		IF nCntHybridDispenser = cMaxHybridDispenser THEN	//maximale Anzahl des spez.Objecttypes erreicht, Object kann nicht angelegt werden
			M_CreateObject := E_ErrorIdObjMgmt.ERRORID_CntHybridDispenserExceeded;	//Rückgabe Error
			RETURN;
		ELSE
			nCntHybridDispenser := nCntHybridDispenser + 1;
			a_pObjects[nObjectID] := ADR(afbHybridDispenser[nCntHybridDispenser]);
			afbHybridDispenser[nCntHybridDispenser].P_nObjectID := nObjectID;
			nCntNotifiIds := nCntNotifiIds + 1;
			afbHybridDispenser[nCntHybridDispenser].P_nNotifyId := nCntNotifiIds;
			nNotifyId := nCntNotifiIds;
		END_IF
		
	E_ObjectType.OBJECTTYPE_DeloDot:
		IF nCntDeloDot = cMaxDeloDots THEN	//maximale Anzahl des spez.Objecttypes erreicht, Object kann nicht angelegt werden
			M_CreateObject := E_ErrorIdObjMgmt.ERRORID_CntDeloDotsExceeded;	//Rückgabe Error
			RETURN;
		ELSE
			nCntDeloDot := nCntDeloDot + 1;
			a_pObjects[nObjectID] := ADR(afbDeloDot[nCntDeloDot]);
			afbDeloDot[nCntDeloDot].P_nObjectID := nObjectID;
			nCntNotifiIds := nCntNotifiIds + 1;
			afbDeloDot[nCntDeloDot].P_nNotifyId := nCntNotifiIds;
			nNotifyId := nCntNotifiIds;
		END_IF

	E_ObjectType.OBJECTTYPE_Diluter:
		IF nCntDiluter = cMaxDiluters THEN	//maximale Anzahl des spez.Objecttypes erreicht, Object kann nicht angelegt werden
			M_CreateObject := E_ErrorIdObjMgmt.ERRORID_CntDilutersExceeded;	//Rückgabe Error
			RETURN;
		ELSE
			nCntDiluter := nCntDiluter + 1;
			a_pObjects[nObjectID] := ADR(afbDiluter[nCntDiluter]);
			afbDiluter[nCntDiluter].P_nObjectID := nObjectID;
			nCntNotifiIds := nCntNotifiIds + 1;
			afbDiluter[nCntDiluter].P_nNotifyId := nCntNotifiIds;
			nNotifyId := nCntNotifiIds;
		END_IF
		
	E_ObjectType.OBJECTTYPE_Diluter3Inputs:
		IF nCntDiluter3Inputs = cMaxDiluters3Inputs THEN	//maximale Anzahl des spez.Objecttypes erreicht, Object kann nicht angelegt werden
			M_CreateObject := E_ErrorIdObjMgmt.ERRORID_CntDilutersExceeded;	//Rückgabe Error
			RETURN;
		ELSE
			nCntDiluter3Inputs := nCntDiluter3Inputs + 1;
			a_pObjects[nObjectID] := ADR(afbDiluter3Inputs[nCntDiluter3Inputs]);
			afbDiluter3Inputs[nCntDiluter3Inputs].P_nObjectID := nObjectID;
			nCntNotifiIds := nCntNotifiIds + 1;
			afbDiluter3Inputs[nCntDiluter3Inputs].P_nNotifyId := nCntNotifiIds;
			nNotifyId := nCntNotifiIds;
		END_IF
		
	E_ObjectType.OBJECTTYPE_DryPad:
		IF nCntDrayPad = cMaxDrayPads THEN	//maximale Anzahl des spez.Objecttypes erreicht, Object kann nicht angelegt werden
			M_CreateObject := E_ErrorIdObjMgmt.ERRORID_CntDrayPadsExceeded;	//Rückgabe Error
			RETURN;
		ELSE
			nCntDrayPad := nCntDrayPad + 1;
			a_pObjects[nObjectID] := ADR(afbDryPad[nCntDrayPad]);
			afbDryPad[nCntDrayPad].P_nObjectID := nObjectID;
			nCntNotifiIds := nCntNotifiIds + 1;
			afbDryPad[nCntDrayPad].P_nNotifyId := nCntNotifiIds;
			nNotifyId := nCntNotifiIds;
		END_IF
		
	E_ObjectType.OBJECTTYPE_DummyTool:
		IF nCntDummyTool = cMaxDummyTools THEN	//maximale Anzahl des spez.Objecttypes erreicht, Object kann nicht angelegt werden
			M_CreateObject := E_ErrorIdObjMgmt.ERRORID_CntDummyToolExceeded;	//Rückgabe Error
			RETURN;
		ELSE
			nCntDummyTool := nCntDummyTool + 1;
			a_pObjects[nObjectID] := ADR(afbDummyTool[nCntDummyTool]);
			afbDummyTool[nCntDummyTool].P_nObjectID := nObjectID;
			nCntNotifiIds := nCntNotifiIds + 1;
			afbDummyTool[nCntDummyTool].P_nNotifyId := nCntNotifiIds;
			nNotifyId := nCntNotifiIds;
 		END_IF		
		
	E_ObjectType.OBJECTTYPE_Exposure:
		IF nCntExposure = cMaxExposure THEN	//maximale Anzahl des spez.Objecttypes erreicht, Object kann nicht angelegt werden
			M_CreateObject := E_ErrorIdObjMgmt.ERRORID_CntExposureExceeded;	//Rückgabe Error
			RETURN;
		ELSE
			nCntExposure := nCntExposure + 1;
			a_pObjects[nObjectID] := ADR(afbExposure[nCntExposure]);
			afbExposure[nCntExposure].P_nObjectID := nObjectID;
			nCntNotifiIds := nCntNotifiIds + 1;
			afbExposure[nCntExposure].P_nNotifyId := nCntNotifiIds;
			nNotifyId := nCntNotifiIds;
		END_IF
		
	E_ObjectType.OBJECTTYPE_Extruder:
		IF nCntExtruder = cMaxExtruder THEN	//maximale Anzahl des spez.Objecttypes erreicht, Object kann nicht angelegt werden
			M_CreateObject := E_ErrorIdObjMgmt.ERRORID_CntExtruderExceeded;	//Rückgabe Error
			RETURN;
		ELSE
			nCntExtruder := nCntExtruder + 1;
			a_pObjects[nObjectID] := ADR(afbExtruder[nCntExtruder]);
			afbExtruder[nCntExtruder].P_nObjectID := nObjectID;
			nCntNotifiIds := nCntNotifiIds + 1;
			afbExtruder[nCntExtruder].P_nNotifyId := nCntNotifiIds;
			nNotifyId := nCntNotifiIds;
		END_IF	
		
	E_ObjectType.OBJECTTYPE_FlipTube:
			pFlipTube := __NEW(FB_FlipTube);
			pFlipTube^.P_nObjectID := nObjectID;
			a_pObjects[nObjectID] := pFlipTube;	
		
	E_ObjectType.OBJECTTYPE_FlipTubeHandler:	//FlipTubeHandler
		IF nCntFlipTubeHandler = cMaxFlipTubeHandler THEN	//maximale Anzahl des spez.Objecttypes erreicht, Object kann nicht angelegt werden
			M_CreateObject := E_ErrorIdObjMgmt.ERRORID_CntFlipTubePinExceeded;	//Rückgabe Error
			RETURN;
		ELSE
			nCntFlipTubeHandler := nCntFlipTubeHandler + 1;
			a_pObjects[nObjectID] := ADR(afbFlipTubeHandler[nCntFlipTubeHandler]);
			afbFlipTubeHandler[nCntFlipTubeHandler].P_nObjectID := nObjectID;
			nCntNotifiIds := nCntNotifiIds + 1;
			afbFlipTubeHandler[nCntFlipTubeHandler].P_nNotifyId := nCntNotifiIds;
			nNotifyId := nCntNotifiIds;
		END_IF
		
	E_ObjectType.OBJECTTYPE_FlipTubeRack:
		IF nCntFlipTubeRack = cMaxFlipTubeRack THEN	//maximale Anzahl des spez.Objecttypes erreicht, Object kann nicht angelegt werden
			M_CreateObject := E_ErrorIdObjMgmt.ERRORID_CntFlipTubeRackExceeded;	//Rückgabe Error
			RETURN;
		ELSE
			nCntFlipTubeRack := nCntFlipTubeRack + 1;
			a_pObjects[nObjectID] := ADR(afbFlipTubeRack[nCntFlipTubeRack]);
			afbFlipTubeRack[nCntFlipTubeRack].P_nObjectID := nObjectID;
		END_IF
		
	E_ObjectType.OBJECTTYPE_Gripper:
		IF nCntGripper = cMaxGripper THEN	//maximale Anzahl des spez.Objecttypes erreicht, Object kann nicht angelegt werden
			M_CreateObject := E_ErrorIdObjMgmt.ERRORID_CntGripperExceeded;	//Rückgabe Error
			RETURN;
		ELSE
			nCntGripper := nCntGripper + 1;
			a_pObjects[nObjectID] := ADR(afbGripper[nCntGripper]);
			afbGripper[nCntGripper].P_nObjectID := nObjectID;
			nCntNotifiIds := nCntNotifiIds + 1;
			afbGripper[nCntGripper].P_nNotifyId := nCntNotifiIds;
			nNotifyId := nCntNotifiIds;
		END_IF
		
	E_ObjectType.OBJECTTYPE_HighVoltTray:
		IF nCntHighVoltTray = cMaxHighVoltTray THEN	//maximale Anzahl des spez.Objecttypes erreicht, Object kann nicht angelegt werden
			M_CreateObject := E_ErrorIdObjMgmt.ERRORID_CntHighVoltTrayExceeded;	//Rückgabe Error
			RETURN;
		ELSE
			nCntHighVoltTray := nCntHighVoltTray + 1;
			a_pObjects[nObjectID] := ADR(afbHighVoltTray[nCntHighVoltTray]);
			afbHighVoltTray[nCntHighVoltTray].P_nObjectID := nObjectID;
			nCntNotifiIds := nCntNotifiIds + 1;
			afbHighVoltTray[nCntHighVoltTray].P_nNotifyId := nCntNotifiIds;			
			nNotifyId := nCntNotifiIds;
		END_IF
		
	E_ObjectType.OBJECTTYPE_InkStation:
		IF nCntInkStation = cMaxInkStations THEN	//maximale Anzahl des spez.Objecttypes erreicht, Object kann nicht angelegt werden
			M_CreateObject := E_ErrorIdObjMgmt.ERRORID_CntInkStationsExceeded;	//Rückgabe Error
			RETURN;
		ELSE
			nCntInkStation := nCntInkStation + 1;
			a_pObjects[nObjectID] := ADR(afbInkStation[nCntInkStation]);
			afbInkStation[nCntInkStation].P_nObjectID := nObjectID;
			nCntNotifiIds := nCntNotifiIds + 1;
			afbInkStation[nCntInkStation].P_nNotifyId := nCntNotifiIds;			
			nNotifyId := nCntNotifiIds;
		END_IF
		
	E_ObjectType.OBJECTTYPE_LiquidReserve:
		IF nCntLiquidReserve = cMaxLiquidReserve THEN	//maximale Anzahl des spez.Objecttypes erreicht, Object kann nicht angelegt werden
			M_CreateObject := E_ErrorIdObjMgmt.ERRORID_Cnt4LiquidReserveExceeded;	//Rückgabe Error
			RETURN;
		ELSE
			nCntLiquidReserve := nCntLiquidReserve + 1;
			a_pObjects[nObjectID] := ADR(afbLiquidReserve[nCntLiquidReserve]);
			afbLiquidReserve[nCntLiquidReserve].P_nObjectID := nObjectID;
			nCntNotifiIds := nCntNotifiIds + 1;
			afbLiquidReserve[nCntLiquidReserve].P_nNotifyId := nCntNotifiIds;
			nNotifyId := nCntNotifiIds;
		END_IF
		
	E_ObjectType.OBJECTTYPE_Luer:
		IF nCntLuer = cMaxLuer THEN	//maximale Anzahl des spez.Objecttypes erreicht, Object kann nicht angelegt werden
			M_CreateObject := E_ErrorIdObjMgmt.ERRORID_CntLuerExceeded;	//Rückgabe Error
			RETURN;
		ELSE
			nCntLuer := nCntLuer + 1;
			a_pObjects[nObjectID] := ADR(afbLuer[nCntLuer]);
			afbLuer[nCntLuer].P_nObjectID := nObjectID;
			nCntNotifiIds := nCntNotifiIds + 1;
			afbLuer[nCntLuer].P_nNotifyId := nCntNotifiIds;
			nNotifyId := nCntNotifiIds;
		END_IF
		
	E_ObjectType.OBJECTTYPE_Mtp:
		pMtp := __NEW(FB_Mtp);
		pMtp^.P_nObjectID := nObjectID;
		a_pObjects[nObjectID] := pMtp;
		
	E_ObjectType.OBJECTTYPE_MtpHolder:		//MTP-Holder
		IF nCntMtpHolder = cMaxMtpHolders THEN	//maximale Anzahl des spez.Objecttypes erreicht, Object kann nicht angelegt werden
			M_CreateObject := E_ErrorIdObjMgmt.ERRORID_CntMtpHoldersExceeded;	//Rückgabe Error
			RETURN;
		ELSE
			nCntMtpHolder := nCntMtpHolder + 1;
			a_pObjects[nObjectID] := ADR(afbMtpHolder[nCntMtpHolder]);
			afbMtpHolder[nCntMtpHolder].P_nObjectID := nObjectID;
			nCntNotifiIds := nCntNotifiIds + 1;
			afbMtpHolder[nCntMtpHolder].P_nNotifyId := nCntNotifiIds;
			nNotifyId := nCntNotifiIds;
		END_IF	
		
	E_ObjectType.OBJECTTYPE_MZHead:
		IF nCntMZHead = cMaxMzHeads THEN	//maximale Anzahl des spez.Objecttypes erreicht, Object kann nicht angelegt werden
			M_CreateObject := E_ErrorIdObjMgmt.ERRORID_CntMZHeadsExceeded;	//Rückgabe Error
			RETURN;
		ELSE
			nCntMZHead := nCntMZHead + 1;
			a_pObjects[nObjectID] := ADR(afbMzHead[nCntMZHead]);
			afbMzHead[nCntMZHead].P_nObjectID := nObjectID;
			nCntNotifiIds := nCntNotifiIds + 1;
			afbMzHead[nCntMZHead].P_nNotifyId := nCntNotifiIds; 
			nNotifyId := nCntNotifiIds; 
		END_IF
		
	E_ObjectType.OBJECTTYPE_Needle:
		pNeedle := __NEW(FB_Needle);
		pNeedle^.P_nObjectID := nObjectID;
		a_pObjects[nObjectID] := pNeedle;	
		
	E_ObjectType.OBJECTTYPE_NeedleRack:
		IF nCntNeedleRack = cMaxNeedleRack THEN	//maximale Anzahl des spez.Objecttypes erreicht, Object kann nicht angelegt werden
			M_CreateObject := E_ErrorIdObjMgmt.ERRORID_CntNeedleRackExceeded;	//Rückgabe Error
			RETURN;
		ELSE
			nCntNeedleRack := nCntNeedleRack + 1;
			a_pObjects[nObjectID] := ADR(afbNeedleRack[nCntNeedleRack]);
			afbNeedleRack[nCntNeedleRack].P_nObjectID := nObjectID;
		END_IF
		
	E_ObjectType.OBJECTTYPE_Nozzle:
		pNozzle := __NEW(FB_Nozzle);
		pNozzle^.P_nObjectID := nObjectID;
		a_pObjects[nObjectID] := pNozzle;	
	
	E_ObjectType.OBJECTTYPE_TwinPiezoHolder:
		IF nCntTwinPiezoHolder = cMaxTwinPiezoHolder THEN	//maximale Anzahl des spez.Objecttypes erreicht, Object kann nicht angelegt werden
			M_CreateObject := E_ErrorIdObjMgmt.ERRORID_CntTwinPiezoHolderExceeded;	//Rückgabe Error
			RETURN;
		ELSE
			nCntTwinPiezoHolder := nCntTwinPiezoHolder + 1;
			a_pObjects[nObjectID] := ADR(afbTwinPiezoHolder[nCntTwinPiezoHolder]);
			afbTwinPiezoHolder[nCntTwinPiezoHolder].P_nObjectID := nObjectID;
			nCntNotifiIds := nCntNotifiIds + 1;
			afbTwinPiezoHolder[nCntTwinPiezoHolder].P_nNotifyId := nCntNotifiIds;
			nNotifyId := nCntNotifiIds;			
		END_IF
		
	E_ObjectType.OBJECTTYPE_TwinExtruder:
		IF nCntTwinExtruder = cMaxTwinExtruder THEN	//maximale Anzahl des spez.Objecttypes erreicht, Object kann nicht angelegt werden
			M_CreateObject := E_ErrorIdObjMgmt.ERRORID_CntTwinExtruderExceeded;	//Rückgabe Error
			RETURN;
		ELSE
			nCntTwinExtruder := nCntTwinExtruder + 1;
			a_pObjects[nObjectID] := ADR(afbTwinExtruder[nCntTwinExtruder]);
			afbTwinExtruder[nCntTwinExtruder].P_nObjectID := nObjectID;
			nCntNotifiIds := nCntNotifiIds + 1;
			afbTwinExtruder[nCntTwinExtruder].P_nNotifyId := nCntNotifiIds;
			nNotifyId := nCntNotifiIds;			
		END_IF		
		
	E_ObjectType.OBJECTTYPE_SinglePiezoHolder:
		IF nCntSinglePiezoHolder = cMaxSinglePiezoHolder THEN	//maximale Anzahl des spez.Objecttypes erreicht, Object kann nicht angelegt werden
			M_CreateObject := E_ErrorIdObjMgmt.ERRORID_CntSinglePiezoHolderExceeded;	//Rückgabe Error
			RETURN;
		ELSE
			nCntSinglePiezoHolder := nCntSinglePiezoHolder + 1;
			a_pObjects[nObjectID] := ADR(afbSinglePiezoHolder[nCntSinglePiezoHolder]);
			afbSinglePiezoHolder[nCntSinglePiezoHolder].P_nObjectID := nObjectID;
			nCntNotifiIds := nCntNotifiIds + 1;
			afbSinglePiezoHolder[nCntSinglePiezoHolder].P_nNotifyId := nCntNotifiIds;
			nNotifyId := nCntNotifiIds;			
		END_IF
		
	E_ObjectType.OBJECTTYPE_PassivPip:
		IF nCntPassivPip = cMaxPassivPips THEN	//maximale Anzahl des spez.Objecttypes erreicht, Object kann nicht angelegt werden
			M_CreateObject := E_ErrorIdObjMgmt.ERRORID_CntPassivPipsExceeded;	//Rückgabe Error
			RETURN;
		ELSE
			nCntPassivPip := nCntPassivPip + 1;
			a_pObjects[nObjectID] := ADR(afbPassivPip[nCntPassivPip]);
			afbPassivPip[nCntPassivPip].P_nObjectID := nObjectID;
			nCntNotifiIds := nCntNotifiIds + 1;
			afbPassivPip[nCntPassivPip].P_nNotifyId := nCntNotifiIds;
			nNotifyId := nCntNotifiIds;	
		END_IF
		
	E_ObjectType.OBJECTTYPE_pHElectrode:
		IF nCntpHElectrode = cMaxpHElectrodes THEN	//maximale Anzahl des spez.Objecttypes erreicht, Object kann nicht angelegt werden
			M_CreateObject := E_ErrorIdObjMgmt.ERRORID_CntpHElectrodesExceeded;	//Rückgabe Error
			RETURN;
		ELSE
			nCntpHElectrode := nCntpHElectrode + 1;
			a_pObjects[nObjectID] := ADR(afbpHElectrode[nCntpHElectrode]);
			afbpHElectrode[nCntpHElectrode].P_nObjectID := nObjectID;
			nCntNotifiIds := nCntNotifiIds + 1;
			afbpHElectrode[nCntpHElectrode].P_nNotifyId := nCntNotifiIds;
			nNotifyId := nCntNotifiIds;	
		END_IF
		
	E_ObjectType.OBJECTTYPE_pHElectrodeCap:
		pPHElectrodeCap := __NEW(FB_pHElectrodeCap);
		pPHElectrodeCap^.P_nObjectID := nObjectID;
		a_pObjects[nObjectID] := pPHElectrodeCap;		
	
	E_ObjectType.OBJECTTYPE_pHElectrodeCapRack:
		IF nCntpHElectrodeCapRack = cMaxpHElectrodeCapRack THEN	//maximale Anzahl des spez.Objecttypes erreicht, Object kann nicht angelegt werden
			M_CreateObject := E_ErrorIdObjMgmt.ERRORID_CntpHElectrodeCapRacksExceeded;	//Rückgabe Error
			RETURN;
		ELSE
			nCntpHElectrodeCapRack := nCntpHElectrodeCapRack + 1;
			a_pObjects[nObjectID] := ADR(afbpHElectrodeCapRack[nCntpHElectrodeCapRack]);
			afbpHElectrodeCapRack[nCntpHElectrodeCapRack].P_nObjectID := nObjectID;
		END_IF
		
	E_ObjectType.OBJECTTYPE_PickPlacePip:
		IF nCntPickPlacePip = cMaxPickPlacePip THEN	//maximale Anzahl des spez.Objecttypes erreicht, Object kann nicht angelegt werden
			M_CreateObject := E_ErrorIdObjMgmt.ERRORID_CntPickPlacePipExceeded;	//Rückgabe Error
			RETURN;
		ELSE
			nCntPickPlacePip := nCntPickPlacePip + 1;
			a_pObjects[nObjectID] := ADR(afbPickPlacePip[nCntPickPlacePip]);
			afbPickPlacePip[nCntPickPlacePip].P_nObjectID := nObjectID;
			nCntNotifiIds := nCntNotifiIds + 1;
			afbPickPlacePip[nCntPickPlacePip].P_nNotifyId := nCntNotifiIds;
			nNotifyId := nCntNotifiIds;
		END_IF	
		
	E_ObjectType.OBJECTTYPE_PiezoPip:
		IF nCntPiezoPip = cMaxPiezoPips THEN	//maximale Anzahl des spez.Objecttypes erreicht, Object kann nicht angelegt werden
			M_CreateObject := E_ErrorIdObjMgmt.ERRORID_CntPiezoPipsExceeded;	//Rückgabe Error
			RETURN;
		ELSE
			nCntPiezoPip := nCntPiezoPip + 1;
			a_pObjects[nObjectID] := ADR(afbPiezoPip[nCntPiezoPip]);
			afbPiezoPip[nCntPiezoPip].P_nObjectID := nObjectID;
			nCntNotifiIds := nCntNotifiIds + 1;
			afbPiezoPip[nCntPiezoPip].P_nNotifyId := nCntNotifiIds;
			nNotifyId := nCntNotifiIds;
		END_IF

	E_ObjectType.OBJECTTYPE_Point:
		pPoint := __NEW(FB_Point);
		pPoint^.P_nObjectID := nObjectID;
		a_pObjects[nObjectID] := pPoint;
		
	E_ObjectType.OBJECTTYPE_Port:
		pPort := __NEW(FB_Port);
		pPort^.P_nObjectID := nObjectID;
		a_pObjects[nObjectID] := pPort;
		
	E_ObjectType.OBJECTTYPE_PortRack:
		IF nCntPortRack = cMaxPortRack THEN	//maximale Anzahl des spez.Objecttypes erreicht, Object kann nicht angelegt werden
			M_CreateObject := E_ErrorIdObjMgmt.ERRORID_CntPortRackExceeded;	//Rückgabe Error
			RETURN;
		ELSE
			nCntPortRack := nCntPortRack + 1;
			a_pObjects[nObjectID] := ADR(afbPortRack[nCntPortRack]);
			afbPortRack[nCntPortRack].P_nObjectID := nObjectID;
		END_IF			
		
	E_ObjectType.OBJECTTYPE_PowderPip: //Pulverpipette
		IF nCntPowderPip = cMaxPowderPips THEN	//maximale Anzahl des spez.Objecttypes erreicht, Object kann nicht angelegt werden
			M_CreateObject := E_ErrorIdObjMgmt.ERRORID_CntPowderPipsExceeded;	//Rückgabe Error
			RETURN;
		ELSE
			nCntPowderPip := nCntPowderPip + 1;
			a_pObjects[nObjectID] := ADR(afbPowderPip[nCntPowderPip]);
			afbPowderPip[nCntPowderPip].P_nObjectID := nObjectID;
			nCntNotifiIds := nCntNotifiIds + 1;
			afbPowderPip[nCntPowderPip].P_nNotifyId := nCntNotifiIds;
			nNotifyId := nCntNotifiIds;			
		END_IF	
		
	E_ObjectType.OBJECTTYPE_PowderStation:
		IF nCntPowderStation = cMaxPowderStations THEN	//maximale Anzahl des spez.Objecttypes erreicht, Object kann nicht angelegt werden
			M_CreateObject := E_ErrorIdObjMgmt.ERRORID_CntPowderStationsExceeded;	//Rückgabe Error
			RETURN;
		ELSE
			nCntPowderStation := nCntPowderStation + 1;
			a_pObjects[nObjectID] := ADR(afbPowderStation[nCntPowderStation]);
			afbPowderStation[nCntPowderStation].P_nObjectID := nObjectID;
			nCntNotifiIds := nCntNotifiIds + 1;
			afbPowderStation[nCntPowderStation].P_nNotifyId := nCntNotifiIds;
			nNotifyId := nCntNotifiIds;
		END_IF
		
	E_ObjectType.OBJECTTYPE_Reactor:
		IF nCntReactor = cMaxReactors THEN	//maximale Anzahl des spez.Objecttypes erreicht, Object kann nicht angelegt werden
			M_CreateObject := E_ErrorIdObjMgmt.ERRORID_CntReactorExceeded;	//Rückgabe Error
			RETURN;
		ELSE
			nCntReactor := nCntReactor + 1;
			a_pObjects[nObjectID] := ADR(afbReactor[nCntReactor]);
			afbReactor[nCntReactor].P_nObjectID := nObjectID;
			nCntNotifiIds := nCntNotifiIds + 1;
			afbReactor[nCntReactor].P_nNotifyId := nCntNotifiIds;
			nNotifyId := nCntNotifiIds;
		END_IF
			
	E_ObjectType.OBJECTTYPE_Septum:
		pSeptum := __NEW(FB_Septum);
		pSeptum^.P_nObjectID := nObjectID;
		a_pObjects[nObjectID] := pSeptum;	
	
	E_ObjectType.OBJECTTYPE_SeptumRack:
		IF nCntSeptumRack = cMaxSeptumRack THEN	//maximale Anzahl des spez.Objecttypes erreicht, Object kann nicht angelegt werden
			M_CreateObject := E_ErrorIdObjMgmt.ERRORID_CntSeptumRackExceeded;	//Rückgabe Error
			RETURN;
		ELSE
			nCntSeptumRack := nCntSeptumRack + 1;
			a_pObjects[nObjectID] := ADR(afbSeptumRack[nCntSeptumRack]);
			afbSeptumRack[nCntSeptumRack].P_nObjectID := nObjectID;
		END_IF			
		
	E_ObjectType.OBJECTTYPE_SeptumWaste:
		IF nCntSeptumWaste = cMaxSeptumWaste THEN	//maximale Anzahl des spez.Objecttypes erreicht, Object kann nicht angelegt werden
			M_CreateObject := E_ErrorIdObjMgmt.ERRORID_CntSeptumWasteExceeded;	//Rückgabe Error
			RETURN;
		ELSE
			nCntSeptumWaste := nCntSeptumWaste + 1;
			a_pObjects[nObjectID] := ADR(afbSeptumWaste[nCntSeptumWaste]);
			afbSeptumWaste[nCntSeptumWaste].P_nObjectID := nObjectID;
		END_IF		

	E_ObjectType.OBJECTTYPE_Slide:
		pSlide := __NEW(FB_Slide);
		pSlide^.P_nObjectID := nObjectID;
		a_pObjects[nObjectID] := pSlide;
	
	E_ObjectType.OBJECTTYPE_SpotArray:
		pSpotArray := __NEW(FB_SpotArray);
		pSpotArray^.P_nObjectID := nObjectID;
		a_pObjects[nObjectID] := pSpotArray;	
	
	(*
	E_ObjectType.OBJECTTYPE_SpotPattern:
		pSpotPattern := __NEW(FB_SpotPattern);
		pSpotPattern^.P_nObjectID := nObjectID;
		a_pObjects[nObjectID] := pSpotPattern;	*)
	
	E_ObjectType.OBJECTTYPE_Stamp:
		pStamp := __NEW(FB_Stamp);
		pStamp^.P_nObjectID := nObjectID;
		a_pObjects[nObjectID] := pStamp;
		
	E_ObjectType.OBJECTTYPE_StampMagazine:
		IF nCntStampMagazine = cMaxStampMagazines THEN	//maximale Anzahl des spez.Objecttypes erreicht, Object kann nicht angelegt werden
			M_CreateObject := E_ErrorIdObjMgmt.ERRORID_CntStampHoldersExceeded;	//Rückgabe Error
			RETURN;
		ELSE
			nCntStampMagazine := nCntStampMagazine + 1;
			a_pObjects[nObjectID] := ADR(afbStampMagazine[nCntStampMagazine]);
			afbStampMagazine[nCntStampMagazine].P_nObjectID := nObjectID;
		END_IF

	E_ObjectType.OBJECTTYPE_StampSupport:
		IF nCntStampSupport = cMaxStampSupports THEN	//maximale Anzahl des spez.Objecttypes erreicht, Object kann nicht angelegt werden
			M_CreateObject := E_ErrorIdObjMgmt.ERRORID_CntStampSupportsExceeded;	//Rückgabe Error
			RETURN;
		ELSE
			nCntStampSupport := nCntStampSupport + 1;
			a_pObjects[nObjectID] := ADR(afbStampSupport[nCntStampSupport]);
			afbStampSupport[nCntStampSupport].P_nObjectID := nObjectID;
			nCntNotifiIds := nCntNotifiIds + 1;
			afbStampSupport[nCntStampSupport].P_nNotifyId := nCntNotifiIds;
			nNotifyId := nCntNotifiIds;
		END_IF
	
	E_ObjectType.OBJECTTYPE_Stroboscope:
		IF nCntStroboscope = cMaxStroboscopes THEN	//maximale Anzahl des spez.Objecttypes erreicht, Object kann nicht angelegt werden
			M_CreateObject := E_ErrorIdObjMgmt.ERRORID_CntStroboscopesExceeded;	//Rückgabe Error
			RETURN;
		ELSE
			nCntStroboscope := nCntStroboscope + 1;
			a_pObjects[nObjectID] := ADR(afbStroboscope[nCntStroboscope]);
			afbStroboscope[nCntStroboscope].P_nObjectID := nObjectID;
			nCntNotifiIds := nCntNotifiIds + 1;
			afbStroboscope[nCntStroboscope].P_nNotifyId := nCntNotifiIds;
			nNotifyId := nCntNotifiIds;	
		END_IF
		
	E_ObjectType.OBJECTTYPE_Stacker:
		IF nCntStacker = cMaxStacker THEN	//maximale Anzahl des spez.Objecttypes erreicht, Object kann nicht angelegt werden
			M_CreateObject := E_ErrorIdObjMgmt.ERRORID_CntStackerExceeded;	//Rückgabe Error
			RETURN;
		ELSE
			nCntStacker := nCntStacker + 1;
			a_pObjects[nObjectID] := ADR(afbStacker[nCntStacker]);
			afbStacker[nCntStacker].P_nObjectID := nObjectID;
			nCntNotifiIds := nCntNotifiIds + 1;
			afbStacker[nCntStacker].P_nNotifyId := nCntNotifiIds;
			nNotifyId := nCntNotifiIds;	
		END_IF
		
	E_ObjectType.OBJECTTYPE_SolenoidPip:
		IF nCntSolenoidPip = cMaxSolenoidPip THEN	//maximale Anzahl des spez.Objecttypes erreicht, Object kann nicht angelegt werden
			M_CreateObject := E_ErrorIdObjMgmt.ERRORID_CntSolenoidPipExceeded;	//Rückgabe Error
			RETURN;
		ELSE
			nCntSolenoidPip := nCntSolenoidPip + 1;
			a_pObjects[nObjectID] := ADR(afbSolenoidPip[nCntSolenoidPip]);
			afbSolenoidPip[nCntSolenoidPip].P_nObjectID := nObjectID;
			nCntNotifiIds := nCntNotifiIds + 1;
			afbSolenoidPip[nCntSolenoidPip].P_nNotifyId := nCntNotifiIds;
			nNotifyId := nCntNotifiIds;
		END_IF	
		
	E_ObjectType.OBJECTTYPE_SubstHolder:
		IF nCntSubstHolder = cMaxSubstHolders THEN	//maximale Anzahl des spez.Objecttypes erreicht, Object kann nicht angelegt werden
			M_CreateObject := E_ErrorIdObjMgmt.ERRORID_CntSubstHoldersExceeded;	//Rückgabe Error
			RETURN;
		ELSE
			nCntSubstHolder := nCntSubstHolder + 1;
			a_pObjects[nObjectID] := ADR(afbSubstHolder[nCntSubstHolder]);
			afbSubstHolder[nCntSubstHolder].P_nObjectID := nObjectID;
			nCntNotifiIds := nCntNotifiIds + 1;
			afbSubstHolder[nCntSubstHolder].P_nNotifyId := nCntNotifiIds;
			nNotifyId := nCntNotifiIds;
		END_IF
		
	E_ObjectType.OBJECTTYPE_SubstHolderUnistat:
		{IF defined(Unistat)}
		IF nCntSubstHolderUnistat = cMaxSubstHolderUnistat THEN	//maximale Anzahl des spez.Objecttypes erreicht, Object kann nicht angelegt werden
			M_CreateObject := E_ErrorIdObjMgmt.ERRORID_CntSubstHoldersExceeded;	//Rückgabe Error
			RETURN;
		ELSE
			nCntSubstHolderUnistat := nCntSubstHolderUnistat + 1;
			a_pObjects[nObjectID] := ADR(afbSubstHolderUnistat[nCntSubstHolderUnistat]);
			afbSubstHolderUnistat[nCntSubstHolderUnistat].P_nObjectID := nObjectID;
			nCntNotifiIds := nCntNotifiIds + 1;
			afbSubstHolderUnistat[nCntSubstHolderUnistat].P_nNotifyId := nCntNotifiIds;
			nNotifyId := nCntNotifiIds;
		END_IF
		{ELSE}
		M_CreateObject := E_ErrorIdObjMgmt.ERRORID_InvalidObjectType;
		RETURN;
		{END_IF}
		
	E_ObjectType.OBJECTTYPE_TargetTray:
			pTray := __NEW(FB_TargetTray);
			pTray^.P_nObjectID := nObjectID;
			a_pObjects[nObjectID] := pTray;
		
	E_ObjectType.OBJECTTYPE_Tip:
			pTip := __NEW(FB_Tip);
			pTip^.P_nObjectID := nObjectID;
			a_pObjects[nObjectID] := pTip;
		
	E_ObjectType.OBJECTTYPE_TipCalibrator:
		IF nCntTipCalibrator = cMaxTipCalibrators THEN	//maximale Anzahl des spez.Objecttypes erreicht, Object kann nicht angelegt werden
			M_CreateObject := E_ErrorIdObjMgmt.ERRORID_CntTipCalibratorExceeded;	//Rückgabe Error
			RETURN;
		ELSE
			nCntTipCalibrator := nCntTipCalibrator + 1;
			a_pObjects[nObjectID] := ADR(afbTipCalibrator[nCntTipCalibrator]);
			afbTipCalibrator[nCntTipCalibrator].P_nObjectID := nObjectID;
			nCntNotifiIds := nCntNotifiIds + 1;
			afbTipCalibrator[nCntTipCalibrator].P_nNotifyId := nCntNotifiIds;
			nNotifyId := nCntNotifiIds;
		END_IF	
		
	E_ObjectType.OBJECTTYPE_TipCleaner:
		IF nCntTipCleaner = cMaxTipCleaners THEN	//maximale Anzahl des spez.Objecttypes erreicht, Object kann nicht angelegt werden
			M_CreateObject := E_ErrorIdObjMgmt.ERRORID_CntTipCleanerExceeded;	//Rückgabe Error
			RETURN;
		ELSE
			nCntTipCleaner := nCntTipCleaner + 1;
			a_pObjects[nObjectID] := ADR(afbTipCleaner[nCntTipCleaner]);
			afbTipCleaner[nCntTipCleaner].P_nObjectID := nObjectID;
			nCntNotifiIds := nCntNotifiIds + 1;
			afbTipCleaner[nCntTipCleaner].P_nNotifyId := nCntNotifiIds;
			nNotifyId := nCntNotifiIds;
		END_IF
		
	E_ObjectType.OBJECTTYPE_TipCleanerGen2:
		IF nCntTipCleanerGen2 = cMaxTipCleanerGen2 THEN	//maximale Anzahl des spez.Objecttypes erreicht, Object kann nicht angelegt werden
			M_CreateObject := E_ErrorIdObjMgmt.ERRORID_CntTipCleanerExceeded;	//Rückgabe Error
			RETURN;
		ELSE
			nCntTipCleanerGen2 := nCntTipCleanerGen2 + 1;
			a_pObjects[nObjectID] := ADR(afbTipCleanerGen2[nCntTipCleanerGen2]);
			afbTipCleanerGen2[nCntTipCleanerGen2].P_nObjectID := nObjectID;
		END_IF
		
	E_ObjectType.OBJECTTYPE_TipRack:
		IF nCntTipRack = cMaxTipRack THEN	//maximale Anzahl des spez.Objecttypes erreicht, Object kann nicht angelegt werden
			M_CreateObject := E_ErrorIdObjMgmt.ERRORID_CntNeedleRackExceeded;	//Rückgabe Error
			RETURN;
		ELSE
			nCntTipRack := nCntTipRack + 1;
			a_pObjects[nObjectID] := ADR(afbTipRack[nCntTipRack]);
			afbTipRack[nCntTipRack].P_nObjectID := nObjectID;
		END_IF

	E_ObjectType.OBJECTTYPE_TitrationTool:
		IF nCntTitrationTool = cMaxTitrationTools THEN	//maximale Anzahl des spez.Objecttypes erreicht, Object kann nicht angelegt werden
			M_CreateObject := E_ErrorIdObjMgmt.ERRORID_CntTitrationToolsExceeded;	//Rückgabe Error
			RETURN;
		ELSE
			nCntTitrationTool := nCntTitrationTool + 1;
			a_pObjects[nObjectID] := ADR(afbTitrationTool[nCntTitrationTool]);
			afbTitrationTool[nCntTitrationTool].P_nObjectID := nObjectID;
			nCntNotifiIds := nCntNotifiIds + 1;
			afbTitrationTool[nCntTitrationTool].P_nNotifyId := nCntNotifiIds;
			nNotifyId := nCntNotifiIds;
 		END_IF

	E_ObjectType.OBJECTTYPE_TrayTransporter:
		IF nCntTrayTransporter = cMaxTrayTransporter THEN	//maximale Anzahl des spez.Objecttypes erreicht, Object kann nicht angelegt werden
			M_CreateObject := E_ErrorIdObjMgmt.ERRORID_CntTrayTransporterExceeded;	//Rückgabe Error
			RETURN;
		ELSE
			nCntTrayTransporter := nCntTrayTransporter + 1;
			a_pObjects[nObjectID] := ADR(afbTrayTransporter[nCntTrayTransporter]);
			afbTrayTransporter[nCntTrayTransporter].P_nObjectID := nObjectID;
			nCntNotifiIds := nCntNotifiIds + 1;
			afbTrayTransporter[nCntTrayTransporter].P_nNotifyId := nCntNotifiIds;
			nNotifyId := nCntNotifiIds;
		END_IF
	
	E_ObjectType.OBJECTTYPE_TriplePip:
		IF nCntTriplePip = cMaxTriplePip THEN	//maximale Anzahl des spez.Objecttypes erreicht, Object kann nicht angelegt werden
			M_CreateObject := E_ErrorIdObjMgmt.ERRORID_CntTriplePipExceeded;	//Rückgabe Error
			RETURN;
		ELSE
			nCntTriplePip := nCntTriplePip + 1;
			a_pObjects[nObjectID] := ADR(afbTriplePip[nCntTriplePip]);
			afbTriplePip[nCntTriplePip].P_nObjectID := nObjectID;
			nCntNotifiIds := nCntNotifiIds + 1;
			afbTriplePip[nCntTriplePip].P_nNotifyId := nCntNotifiIds;
			nNotifyId := nCntNotifiIds;
		END_IF
		
	E_ObjectType.OBJECTTYPE_VacuumHandler:
		IF nCntVacuumHandler = cMaxVacuumHandler THEN	//maximale Anzahl des spez.Objecttypes erreicht, Object kann nicht angelegt werden
			M_CreateObject := E_ErrorIdObjMgmt.ERRORID_CntVacuumHandlerExceeded;	//Rückgabe Error
			RETURN;
		ELSE
			nCntVacuumHandler := nCntVacuumHandler + 1;
			a_pObjects[nObjectID] := ADR(afbVacuumHandler[nCntVacuumHandler]);
			afbVacuumHandler[nCntVacuumHandler].P_nObjectID := nObjectID;
			nCntNotifiIds := nCntNotifiIds + 1;
			afbVacuumHandler[nCntVacuumHandler].P_nNotifyId := nCntNotifiIds;
			nNotifyId := nCntNotifiIds;
		END_IF		
		
	E_ObjectType.OBJECTTYPE_VermesDisp:
		IF nCntVermesDisp = cMaxVermesDisp THEN	//maximale Anzahl des spez.Objecttypes erreicht, Object kann nicht angelegt werden
			M_CreateObject := E_ErrorIdObjMgmt.ERRORID_CntVermesDispExceeded;	//Rückgabe Error
			RETURN;
		ELSE
			nCntVermesDisp := nCntVermesDisp + 1;
			a_pObjects[nObjectID] := ADR(afbVermesDisp[nCntVermesDisp]);
			afbVermesDisp[nCntVermesDisp].P_nObjectID := nObjectID;
			nCntNotifiIds := nCntNotifiIds + 1;
			afbVermesDisp[nCntVermesDisp].P_nNotifyId := nCntNotifiIds;
			nNotifyId := nCntNotifiIds;
 		END_IF

	E_ObjectType.OBJECTTYPE_Vial:
			pVial := __NEW(FB_Vial);
			pVial^.P_nObjectID := nObjectID;
			a_pObjects[nObjectID] := pVial;	
		
	E_ObjectType.OBJECTTYPE_VialClosed:
			pVialClosed := __NEW(FB_VialClosed);
			pVialClosed^.P_nObjectID := nObjectID;
			a_pObjects[nObjectID] := pVialClosed;	
		
	E_ObjectType.OBJECTTYPE_VialRack:
		IF nCntVialRack = cMaxVialRack THEN	//maximale Anzahl des spez.Objecttypes erreicht, Object kann nicht angelegt werden
			M_CreateObject := E_ErrorIdObjMgmt.ERRORID_CntVialRackExceeded;	//Rückgabe Error
			RETURN;
		ELSE
			nCntVialRack := nCntVialRack + 1;
			a_pObjects[nObjectID] := ADR(afbVialRack[nCntVialRack]);
			afbVialRack[nCntVialRack].P_nObjectID := nObjectID;
		END_IF
		
	E_ObjectType.OBJECTTYPE_VialRackClosed:
		IF nCntVialRack = cMaxVialRack THEN	//maximale Anzahl des spez.Objecttypes erreicht, Object kann nicht angelegt werden
			M_CreateObject := E_ErrorIdObjMgmt.ERRORID_CntVialRackExceeded;	//Rückgabe Error
			RETURN;
		ELSE
			nCntVialRack := nCntVialRack + 1;
			a_pObjects[nObjectID] := ADR(afbVialRack[nCntVialRack]);
			afbVialRack[nCntVialRack].P_nObjectID := nObjectID;
			afbVialRack[nCntVialRack].M_OverrideObjectType();
		END_IF		
		
	(*E_ObjectType.OBJECTTYPE_Wafer:
		pWafer := __NEW(FB_Wafer);
		pWafer^.P_nObjectID := nObjectID;
		a_pObjects[nObjectID] := pWafer;*)
		
	E_ObjectType.OBJECTTYPE_WashStation:
		IF nCntWashStation = cMaxWashStations THEN	//maximale Anzahl des spez.Objecttypes erreicht, Object kann nicht angelegt werden
			M_CreateObject := E_ErrorIdObjMgmt.ERRORID_CntWashStationsExceeded;	//Rückgabe Error
			RETURN;
		ELSE
			nCntWashStation := nCntWashStation + 1;
			a_pObjects[nObjectID] := ADR(afbWashStation[nCntWashStation]);
			afbWashStation[nCntWashStation].P_nObjectID := nObjectID;
			nCntNotifiIds := nCntNotifiIds + 1;
			afbWashStation[nCntWashStation].P_nNotifyId := nCntNotifiIds;
			nNotifyId := nCntNotifiIds;
		END_IF
		
	E_ObjectType.OBJECTTYPE_Workplate:
		IF nCntWorkplate = cMaxWorkplates THEN	//maximale Anzahl des spez.Objecttypes erreicht, Object kann nicht angelegt werden
			M_CreateObject := E_ErrorIdObjMgmt.ERRORID_CntWorkplatesExceeded;	//Rückgabe Error
			RETURN;
		ELSE
			nCntWorkplate := nCntWorkplate + 1;
			a_pObjects[nObjectID] := ADR(afbWorkplate[nCntWorkplate]);
			afbWorkplate[nCntWorkplate].P_nObjectID := nObjectID;
		END_IF
		
	E_ObjectType.OBJECTTYPE_WorkplateCamera:
		IF nCntWorkplateCamera = cMaxWorkplateCameras THEN	//maximale Anzahl des spez.Objecttypes erreicht, Object kann nicht angelegt werden
			M_CreateObject := E_ErrorIdObjMgmt.ERRORID_CntWorkplateCameraExceeded;	//Rückgabe Error
			RETURN;
		ELSE
			nCntWorkplateCamera := nCntWorkplateCamera + 1;
			a_pObjects[nObjectID] := ADR(afbWorkplateCamera[nCntWorkplateCamera]);
			afbWorkplateCamera[nCntWorkplateCamera].P_nObjectID := nObjectID;
			nCntNotifiIds := nCntNotifiIds + 1;
			afbWorkplateCamera[nCntWorkplateCamera].P_nNotifyId := nCntNotifiIds;
			nNotifyId := nCntNotifiIds;	
		END_IF		
		
	E_ObjectType.OBJECTTYPE_ZSensor:
		IF nCntZLevelSensor = cMaxZLevelSensors THEN	//maximale Anzahl des spez.Objecttypes erreicht, Object kann nicht angelegt werden
			M_CreateObject := E_ErrorIdObjMgmt.ERRORID_CntZLevelSensorsExceeded;	//Rückgabe Error
			RETURN;
		ELSE
			nCntZLevelSensor := nCntZLevelSensor + 1;
			a_pObjects[nObjectID] := ADR(afbZLevelSensor[nCntZLevelSensor]);
			afbZLevelSensor[nCntZLevelSensor].P_nObjectID := nObjectID;
			nCntNotifiIds := nCntNotifiIds + 1;
			afbZLevelSensor[nCntZLevelSensor].P_nNotifyId := nCntNotifiIds;
			nNotifyId := nCntNotifiIds;
 		END_IF
ELSE
	M_CreateObject := E_ErrorIdObjMgmt.ERRORID_InvalidObjectType;
	RETURN;
END_CASE
nCntObject := nCntObject + 1;

//ParentObject ermitteln aus data[0]
nParentObjectId := DINT_TO_UINT(refCmdData.n32Data[0]);
IF nParentObjectId = 0 THEN	//Soll kein Parent erhalten, nur für Diluter, Workplate und Head zulässig
	IF a_pObjects[nObjectID]^.P_eObjectType = E_ObjectType.OBJECTTYPE_Diluter OR
			a_pObjects[nObjectID]^.P_eObjectType = E_ObjectType.OBJECTTYPE_Diluter3Inputs OR
				a_pObjects[nObjectID]^.P_eObjectType = E_ObjectType.OBJECTTYPE_Workplate OR
					a_pObjects[nObjectID]^.P_eObjectType = E_ObjectType.OBJECTTYPE_MZHead OR
					a_pObjects[nObjectID]^.P_eObjectType = E_ObjectType.OBJECTTYPE_Stacker THEN
					
		a_pObjects[nObjectID]^.P_pObjCollectNode := objectList.M_AddNewNode(a_pObjects[nObjectID],nIndex);
	ELSE
		//Objekttyp muss zwingend an ein Parent
		M_CreateObject := E_ErrorIdObjMgmt.ERRORID_ObjectMustHaveAParent;
	END_IF
ELSIF nParentObjectId > 0 AND nParentObjectId <= cMaxObjects THEN
	pParentObject := a_pObjects[nParentObjectId];
	IF pParentObject > 0 THEN
		nParentSlotNr := DINT_TO_UINT(refCmdData.n32Data[1]);
		M_CreateObject := pParentObject^.M_AddChild(a_pObjects[nObjectID],nParentSlotNr,nIndex);
	ELSE
		M_CreateObject := E_ErrorIdObjMgmt.ERRORID_InvalidParentObject;
	END_IF
ELSE
	M_CreateObject := E_ErrorIdObjMgmt.ERRORID_InvalidParentObject;
END_IF

IF M_CreateObject > 0 THEN
	M_DeleteObject(nObjectID);
ELSE
	M_CreateObject := a_pObjects[nObjectID]^.M_SetAllProps(refCmdData);
	IF M_CreateObject > 0 THEN
		M_DeleteObject(nObjectID);
	ELSE
		refCmdData.aHeader[0] := nObjectID;	//zum Zurücklesen für den GUI-Kernel
		IF a_pObjects[nObjectID]^.M_bIsGroup(E_ObjectGroup.OBJECTGROUP_Device) THEN
			deviceList.M_AddNewNode(a_pObjects[nObjectID],nIndex);
		END_IF
		
		IF a_pObjects[nObjectID]^.M_bIsGroup(E_ObjectGroup.OBJECTGROUP_MzTool) THEN
			fbConfiguration.M_Deactivate();
		END_IF
	END_IF
END_IF
END_METHOD

METHOD M_CustomUnitType2_Error : BOOL
VAR_INPUT
END_VAR

VAR
	i : UINT;
END_VAR
FOR i := 1 TO nCntCustomUnitType2 DO
	 IF afbCustomUnitType2[i].P_bError THEN
		 M_CustomUnitType2_Error := TRUE;
	 END_IF
END_FOR
END_METHOD

METHOD M_DeleteAllObj : E_ErrorIdObjMgmt
VAR_INPUT
END_VAR
VAR
	i		: UINT;
	iter 	: FB_ObjCollectIteratorDeep;
	pObject : POINTER TO FB_Object;
	id 		: UINT;
END_VAR
//Methode zum kompletten Löschen des Objektverzeichnisses

//Objektzählervariablen zurücksetzen
nCntCamera := 0;
nCntCartDispenser := 0;
nCntCartDispStirrer := 0;
nCntCartHolder := 0;
nCntCustomUnitType1 := 0;
nCntCustomUnitType2 := 0;
nCntMultiCartHolder := 0;
nCntHybridDispenser := 0;
nCntDeloDot := 0;	
nCntDiluter := 0;
nCntDiluter3Inputs := 0;
nCntDrayPad := 0;
nCntDummyTool := 0;
nCntExposure := 0;		
nCntFlipTubeHandler	:= 0;			
nCntFlipTubeRack := 0;
nCntGripper := 0;
nCntHighVoltTray := 0;		
nCntInkStation := 0;		
nCntLiquidReserve := 0;			
nCntLuer := 0; 	
nCntMtpHolder := 0;		
nCntMZHead := 0;	
nCntNeedleRack := 0;		
nCntNotifiIds := 0;		
nCntObject := 0;
nCntTwinExtruder := 0;	
nCntTwinPiezoHolder	:= 0;	
nCntPassivPip := 0;
nCntpHElectrode	:= 0;
nCntpHElectrodeCapRack := 0;
nCntPickPlacePip := 0;
nCntPiezoPip := 0;		
nCntPortRack := 0;		
nCntPowderPip := 0;		
nCntPowderStation := 0;			
nCntReactor := 0;	
nCntSampleScan := 0;		
nCntSeptumRack := 0;		
nCntSeptumWaste	:= 0;
nCntSinglePiezoHolder := 0;	
nCntStacker := 0;	
nCntSolenoidPip := 0;
nCntExtruder := 0;
nCntStampMagazine := 0;			
nCntStampSupport := 0;			
nCntStroboscope := 0;		
nCntSubstHolder := 0;
nCntSubstHolderUnistat := 0;
nCntTipCalibrator := 0;			
nCntTipCleaner := 0;
nCntTipCleanerGen2 := 0;
nCntTipRack := 0;
nCntTitrationTool := 0;
nCntTrayTransporter := 0;
nCntTriplePip := 0;		
nCntVacuumHandler := 0;
nCntVermesDisp := 0;			
nCntVialRack := 0;		
nCntWashStation	:= 0;		
nCntWorkplate := 0;
nCntWorkplateCamera := 0;
nCntZLevelSensor := 0;			

